LIN {X 0,Y 523.908,Z 265.034,A -85,B 0,C 180,E1 -4736.634,E2 -4736.634} C_VEL
LIN {X 0,Y 523.939,Z 265.035,A -85,B 0,C 180,E1 -4739.356,E2 -4739.356} C_VEL
LIN {X 0,Y 523.937,Z 265.029,A -85,B 0,C 180,E1 -4742.29,E2 -4742.29} C_VEL
LIN {X 0,Y 523.899,Z 265.041,A -85,B 0,C 180,E1 -4745.427,E2 -4745.427} C_VEL
LIN {X 0,Y 523.983,Z 265.186,A -85,B 0,C 180,E1 -4747.547,E2 -4747.547} C_VEL
LIN {X 0,Y 524.776,Z 271.643,A -85,B 0,C 180,E1 -4748.803,E2 -4748.803} C_VEL
LIN {X 0,Y 524.426,Z 286.9,A -85,B 0,C 180,E1 -4751.644,E2 -4751.644} C_VEL
LIN {X 0,Y 524.115,Z 304.678,A -85,B 0,C 180,E1 -4754.898,E2 -4754.898} C_VEL
LIN {X 0,Y 523.825,Z 322.199,A -85,B 0,C 180,E1 -4758.077,E2 -4758.077} C_VEL
LIN {X 0,Y 524.969,Z 332.235,A -85,B 0,C 180,E1 -4758.254,E2 -4758.254} C_VEL
LIN {X 0,Y 524.703,Z 399.496,A -85,B 0,C 180,E1 -4759.192,E2 -4759.192} C_VEL
LIN {X 0,Y 524.561,Z 409.221,A -85,B 0,C 180,E1 -4759.433,E2 -4759.433} C_VEL
LIN {X 0,Y 524.413,Z 420.832,A -85,B 0,C 180,E1 -4759.869,E2 -4759.869} C_VEL
LIN {X 0,Y 524.207,Z 431.496,A -85,B 0,C 180,E1 -4760.45,E2 -4760.45} C_VEL
LIN {X 0,Y 524.097,Z 439.84,A -85,B 0,C 180,E1 -4761.032,E2 -4761.032} C_VEL
LIN {X 0,Y 523.882,Z 447.732,A -85,B 0,C 180,E1 -4761.708,E2 -4761.708} C_VEL
LIN {X 0,Y 523.71,Z 455.111,A -85,B 0,C 180,E1 -4762.482,E2 -4762.482} C_VEL
LIN {X 0,Y 523.63,Z 462.468,A -85,B 0,C 180,E1 -4763.431,E2 -4763.431} C_VEL
LIN {X 0,Y 523.538,Z 468.474,A -85,B 0,C 180,E1 -4764.415,E2 -4764.415} C_VEL
LIN {X 0,Y 523.406,Z 473.097,A -85,B 0,C 180,E1 -4765.379,E2 -4765.379} C_VEL
LIN {X 0,Y 523.454,Z 476.104,A -85,B 0,C 180,E1 -4766.151,E2 -4766.151} C_VEL
LIN {X 0,Y 523.379,Z 478.431,A -85,B 0,C 180,E1 -4766.921,E2 -4766.921} C_VEL
LIN {X 0,Y 523.336,Z 480.183,A -85,B 0,C 180,E1 -4767.691,E2 -4767.691} C_VEL
LIN {X 0,Y 523.273,Z 481.437,A -85,B 0,C 180,E1 -4768.461,E2 -4768.461} C_VEL
LIN {X 0,Y 523.247,Z 482.217,A -85,B 0,C 180,E1 -4769.23,E2 -4769.23} C_VEL
LIN {X 0,Y 523.246,Z 482.512,A -85,B 0,C 180,E1 -4770,E2 -4770} C_VEL
LIN {X 0,Y 523.247,Z 482.215,A -85,B 0,C 180,E1 -4770.77,E2 -4770.77} C_VEL
LIN {X 0,Y 523.273,Z 481.433,A -85,B 0,C 180,E1 -4771.539,E2 -4771.539} C_VEL
LIN {X 0,Y 523.336,Z 480.177,A -85,B 0,C 180,E1 -4772.309,E2 -4772.309} C_VEL
LIN {X 0,Y 523.407,Z 477.267,A -85,B 0,C 180,E1 -4773.464,E2 -4773.464} C_VEL
LIN {X 0,Y 523.454,Z 474.613,A -85,B 0,C 180,E1 -4774.235,E2 -4774.235} C_VEL
LIN {X 0,Y 523.484,Z 469.419,A -85,B 0,C 180,E1 -4775.392,E2 -4775.392} C_VEL
LIN {X 0,Y 523.596,Z 463.434,A -85,B 0,C 180,E1 -4776.422,E2 -4776.422} C_VEL
LIN {X 0,Y 523.698,Z 456.795,A -85,B 0,C 180,E1 -4777.324,E2 -4777.324} C_VEL
LIN {X 0,Y 523.856,Z 448.738,A -85,B 0,C 180,E1 -4778.195,E2 -4778.195} C_VEL
LIN {X 0,Y 524.08,Z 441.048,A -85,B 0,C 180,E1 -4778.871,E2 -4778.871} C_VEL
LIN {X 0,Y 524.198,Z 432.968,A -85,B 0,C 180,E1 -4779.453,E2 -4779.453} C_VEL
LIN {X 0,Y 524.337,Z 424.594,A -85,B 0,C 180,E1 -4779.937,E2 -4779.937} C_VEL
LIN {X 0,Y 524.502,Z 416.045,A -85,B 0,C 180,E1 -4780.324,E2 -4780.324} C_VEL
LIN {X 0,Y 524.571,Z 405.846,A -85,B 0,C 180,E1 -4780.664,E2 -4780.664} C_VEL
LIN {X 0,Y 524.779,Z 393.965,A -85,B 0,C 180,E1 -4780.904,E2 -4780.904} C_VEL
LIN {X 0,Y 524.782,Z 329.722,A -85,B 0,C 180,E1 -4781.784,E2 -4781.784} C_VEL
LIN {X 0,Y 523.821,Z 322.037,A -85,B 0,C 180,E1 -4781.93,E2 -4781.93} C_VEL
LIN {X 0,Y 524.082,Z 303.651,A -85,B 0,C 180,E1 -4785.231,E2 -4785.231} C_VEL
LIN {X 0,Y 524.369,Z 287.56,A -85,B 0,C 180,E1 -4788.156,E2 -4788.156} C_VEL
LIN {X 0,Y 524.64,Z 270.939,A -85,B 0,C 180,E1 -4791.203,E2 -4791.203} C_VEL
LIN {X 0,Y 523.965,Z 265.034,A -85,B 0,C 180,E1 -4792.349,E2 -4792.349} C_VEL
LIN {X 0,Y 523.896,Z 265.035,A -85,B 0,C 180,E1 -4795.421,E2 -4795.421} C_VEL
LIN {X 0,Y 523.906,Z 265.034,A -85,B 0,C 180,E1 -4798.002,E2 -4798.002} C_VEL
LIN {X 0,Y 523.93,Z 265.037,A -85,B 0,C 180,E1 -4800.852,E2 -4800.852} C_VEL
LIN {X 0,Y 523.924,Z 265.03,A -85,B 0,C 180,E1 -4803.729,E2 -4803.729} C_VEL
LIN {X 0,Y 523.897,Z 265.035,A -85,B 0,C 180,E1 -4806.4,E2 -4806.4} C_VEL
LIN {X 0,Y 523.913,Z 265.041,A -85,B 0,C 180,E1 -4809.084,E2 -4809.084} C_VEL
LIN {X 0,Y 523.931,Z 265.029,A -85,B 0,C 180,E1 -4812.119,E2 -4812.119} C_VEL
LIN {X 0,Y 523.941,Z 265.037,A -85,B 0,C 180,E1 -4815.309,E2 -4815.309} C_VEL
LIN {X 0,Y 523.95,Z 265.026,A -85,B 0,C 180,E1 -4818.689,E2 -4818.689} C_VEL
LIN {X 0,Y 523.903,Z 265.035,A -85,B 0,C 180,E1 -4821.08,E2 -4821.08} C_VEL
LIN {X 0,Y 523.913,Z 265.038,A -85,B 0,C 180,E1 -4823.826,E2 -4823.826} C_VEL
LIN {X 0,Y 523.93,Z 265.027,A -85,B 0,C 180,E1 -4826.635,E2 -4826.635} C_VEL
LIN {X 0,Y 523.944,Z 265.029,A -85,B 0,C 180,E1 -4829.355,E2 -4829.355} C_VEL
LIN {X 0,Y 523.963,Z 265.026,A -85,B 0,C 180,E1 -4832.281,E2 -4832.281} C_VEL
LIN {X 0,Y 523.933,Z 265.03,A -85,B 0,C 180,E1 -4834.58,E2 -4834.58} C_VEL
LIN {X 0,Y 523.905,Z 265.034,A -85,B 0,C 180,E1 -4837.756,E2 -4837.756} C_VEL
LIN {X 0,Y 523.959,Z 265.032,A -85,B 0,C 180,E1 -4840.407,E2 -4840.407} C_VEL
LIN {X 0,Y 523.949,Z 265.027,A -85,B 0,C 180,E1 -4842.837,E2 -4842.837} C_VEL
LIN {X 0,Y 523.96,Z 265.023,A -85,B 0,C 180,E1 -4845.235,E2 -4845.235} C_VEL
LIN {X 0,Y 523.998,Z 265.028,A -85,B 0,C 180,E1 -4848.394,E2 -4848.394} C_VEL
LIN {X 0,Y 523.988,Z 265.019,A -85,B 0,C 180,E1 -4851.516,E2 -4851.516} C_VEL
LIN {X 0,Y 524.083,Z 265.017,A -85,B 0,C 180,E1 -4854.614,E2 -4854.614} C_VEL
LIN {X 0,Y 524.094,Z 265.006,A -85,B 0,C 180,E1 -4857.694,E2 -4857.694} C_VEL
LIN {X 0,Y 524.11,Z 265.012,A -85,B 0,C 180,E1 -4860.768,E2 -4860.768} C_VEL
LIN {X 0,Y 524.059,Z 265.019,A -85,B 0,C 180,E1 -4863.075,E2 -4863.075} C_VEL
LIN {X 0,Y 524.017,Z 265.017,A -85,B 0,C 180,E1 -4866.159,E2 -4866.159} C_VEL
LIN {X 0,Y 523.991,Z 265.02,A -85,B 0,C 180,E1 -4868.484,E2 -4868.484} C_VEL
LIN {X 0,Y 523.988,Z 265.023,A -85,B 0,C 180,E1 -4871.74,E2 -4871.74} C_VEL
LIN {X 0,Y 523.979,Z 265.026,A -85,B 0,C 180,E1 -4875.053,E2 -4875.053} C_VEL
LIN {X 0,Y 523.951,Z 265.031,A -85,B 0,C 180,E1 -4877.97,E2 -4877.97} C_VEL
LIN {X 0,Y 523.959,Z 265.025,A -85,B 0,C 180,E1 -4880.411,E2 -4880.411} C_VEL
LIN {X 0,Y 523.904,Z 265.033,A -85,B 0,C 180,E1 -4882.894,E2 -4882.894} C_VEL
LIN {X 0,Y 523.943,Z 265.031,A -85,B 0,C 180,E1 -4885.419,E2 -4885.419} C_VEL
LIN {X 0,Y 523.96,Z 265.034,A -85,B 0,C 180,E1 -4888,E2 -4888} C_VEL
LIN {X 0,Y 523.939,Z 265.028,A -85,B 0,C 180,E1 -4890.857,E2 -4890.857} C_VEL
LIN {X 0,Y 523.952,Z 265.03,A -85,B 0,C 180,E1 -4893.736,E2 -4893.736} C_VEL
LIN {X 0,Y 523.916,Z 265.039,A -85,B 0,C 180,E1 -4896.406,E2 -4896.406} C_VEL
LIN {X 0,Y 523.923,Z 265.032,A -85,B 0,C 180,E1 -4899.085,E2 -4899.085} C_VEL
LIN {X 0,Y 523.961,Z 265.027,A -85,B 0,C 180,E1 -4901.313,E2 -4901.313} C_VEL
LIN {X 0,Y 523.942,Z 265.155,A -85,B 0,C 180,E1 -4904.015,E2 -4904.015} C_VEL
LIN {X 0,Y 523.901,Z 277.544,A -85,B 0,C 180,E1 -4906.558,E2 -4906.558} C_VEL
LIN {X 0,Y 523.203,Z 280.386,A -85,B 0,C 180,E1 -4907.119,E2 -4907.119} C_VEL
LIN {X 0,Y 517.424,Z 289.883,A -85,B 0,C 180,E1 -4908.932,E2 -4908.932} C_VEL
LIN {X 0,Y 516.76,Z 292.676,A -85,B 0,C 180,E1 -4909.507,E2 -4909.507} C_VEL
LIN {X 0,Y 516.771,Z 294.884,A -85,B 0,C 180,E1 -4909.971,E2 -4909.971} C_VEL
LIN {X 0,Y 518.022,Z 305.126,A -85,B 0,C 180,E1 -4910.155,E2 -4910.155} C_VEL
LIN {X 0,Y 517.74,Z 371.268,A -85,B 0,C 180,E1 -4911.094,E2 -4911.094} C_VEL
LIN {X 0,Y 517.645,Z 381.412,A -85,B 0,C 180,E1 -4911.353,E2 -4911.353} C_VEL
LIN {X 0,Y 517.507,Z 392.694,A -85,B 0,C 180,E1 -4911.791,E2 -4911.791} C_VEL
LIN {X 0,Y 517.283,Z 402.236,A -85,B 0,C 180,E1 -4912.312,E2 -4912.312} C_VEL
LIN {X 0,Y 517.132,Z 410.829,A -85,B 0,C 180,E1 -4912.911,E2 -4912.911} C_VEL
LIN {X 0,Y 516.91,Z 418.134,A -85,B 0,C 180,E1 -4913.534,E2 -4913.534} C_VEL
LIN {X 0,Y 516.803,Z 424.755,A -85,B 0,C 180,E1 -4914.216,E2 -4914.216} C_VEL
LIN {X 0,Y 516.67,Z 430.573,A -85,B 0,C 180,E1 -4914.929,E2 -4914.929} C_VEL
LIN {X 0,Y 516.515,Z 436.787,A -85,B 0,C 180,E1 -4915.857,E2 -4915.857} C_VEL
LIN {X 0,Y 516.448,Z 441.827,A -85,B 0,C 180,E1 -4916.792,E2 -4916.792} C_VEL
LIN {X 0,Y 516.359,Z 446.667,A -85,B 0,C 180,E1 -4917.94,E2 -4917.94} C_VEL
LIN {X 0,Y 516.307,Z 450.049,A -85,B 0,C 180,E1 -4919.044,E2 -4919.044} C_VEL
LIN {X 0,Y 516.239,Z 451.555,A -85,B 0,C 180,E1 -4919.755,E2 -4919.755} C_VEL
LIN {X 0,Y 516.219,Z 452.9,A -85,B 0,C 180,E1 -4920.653,E2 -4920.653} C_VEL
LIN {X 0,Y 516.174,Z 453.582,A -85,B 0,C 180,E1 -4921.541,E2 -4921.541} C_VEL
LIN {X 0,Y 516.179,Z 453.632,A -85,B 0,C 180,E1 -4922.425,E2 -4922.425} C_VEL
LIN {X 0,Y 516.182,Z 453.064,A -85,B 0,C 180,E1 -4923.302,E2 -4923.302} C_VEL
LIN {X 0,Y 516.186,Z 451.886,A -85,B 0,C 180,E1 -4924.172,E2 -4924.172} C_VEL
LIN {X 0,Y 516.267,Z 450.057,A -85,B 0,C 180,E1 -4925.04,E2 -4925.04} C_VEL
LIN {X 0,Y 516.336,Z 447.541,A -85,B 0,C 180,E1 -4925.9,E2 -4925.9} C_VEL
LIN {X 0,Y 516.409,Z 442.393,A -85,B 0,C 180,E1 -4927.179,E2 -4927.179} C_VEL
LIN {X 0,Y 516.515,Z 437.678,A -85,B 0,C 180,E1 -4928.08,E2 -4928.08} C_VEL
LIN {X 0,Y 516.606,Z 432.66,A -85,B 0,C 180,E1 -4928.869,E2 -4928.869} C_VEL
LIN {X 0,Y 516.736,Z 427.232,A -85,B 0,C 180,E1 -4929.585,E2 -4929.585} C_VEL
LIN {X 0,Y 516.891,Z 420.375,A -85,B 0,C 180,E1 -4930.336,E2 -4930.336} C_VEL
LIN {X 0,Y 517.035,Z 413.529,A -85,B 0,C 180,E1 -4930.961,E2 -4930.961} C_VEL
LIN {X 0,Y 517.261,Z 405.127,A -85,B 0,C 180,E1 -4931.586,E2 -4931.586} C_VEL
LIN {X 0,Y 517.429,Z 396.432,A -85,B 0,C 180,E1 -4932.102,E2 -4932.102} C_VEL
LIN {X 0,Y 517.564,Z 387.033,A -85,B 0,C 180,E1 -4932.534,E2 -4932.534} C_VEL
LIN {X 0,Y 517.749,Z 376.5,A -85,B 0,C 180,E1 -4932.88,E2 -4932.88} C_VEL
LIN {X 0,Y 517.852,Z 362.604,A -85,B 0,C 180,E1 -4933.137,E2 -4933.137} C_VEL
LIN {X 0,Y 517.873,Z 302.517,A -85,B 0,C 180,E1 -4933.974,E2 -4933.974} C_VEL
LIN {X 0,Y 516.718,Z 295.169,A -85,B 0,C 180,E1 -4934.115,E2 -4934.115} C_VEL
LIN {X 0,Y 516.912,Z 282.012,A -85,B 0,C 180,E1 -4937.037,E2 -4937.037} C_VEL
LIN {X 0,Y 517.088,Z 269.588,A -85,B 0,C 180,E1 -4939.823,E2 -4939.823} C_VEL
LIN {X 0,Y 516.99,Z 265.9,A -85,B 0,C 180,E1 -4940.71,E2 -4940.71} C_VEL
LIN {X 0,Y 517.003,Z 265.901,A -85,B 0,C 180,E1 -4943.757,E2 -4943.757} C_VEL
LIN {X 0,Y 517.013,Z 265.89,A -85,B 0,C 180,E1 -4946.883,E2 -4946.883} C_VEL
LIN {X 0,Y 517.087,Z 265.889,A -85,B 0,C 180,E1 -4950,E2 -4950} C_VEL
LIN {X 0,Y 517.014,Z 265.89,A -85,B 0,C 180,E1 -4953.117,E2 -4953.117} C_VEL
LIN {X 0,Y 516.99,Z 265.901,A -85,B 0,C 180,E1 -4956.243,E2 -4956.243} C_VEL
LIN {X 0,Y 516.967,Z 265.9,A -85,B 0,C 180,E1 -4958.6,E2 -4958.6} C_VEL
LIN {X 0,Y 516.953,Z 265.9,A -85,B 0,C 180,E1 -4961.806,E2 -4961.806} C_VEL
LIN {X 0,Y 516.946,Z 265.899,A -85,B 0,C 180,E1 -4965.146,E2 -4965.146} C_VEL
LIN {X 0,Y 516.917,Z 265.906,A -85,B 0,C 180,E1 -4968.222,E2 -4968.222} C_VEL
LIN {X 0,Y 516.912,Z 265.912,A -85,B 0,C 180,E1 -4970.701,E2 -4970.701} C_VEL
LIN {X 0,Y 516.901,Z 265.905,A -85,B 0,C 180,E1 -4974.072,E2 -4974.072} C_VEL
LIN {X 0,Y 516.922,Z 265.908,A -85,B 0,C 180,E1 -4976.657,E2 -4976.657} C_VEL
LIN {X 0,Y 516.909,Z 265.905,A -85,B 0,C 180,E1 -4979.523,E2 -4979.523} C_VEL
LIN {X 0,Y 516.891,Z 265.907,A -85,B 0,C 180,E1 -4982.542,E2 -4982.542} C_VEL
LIN {X 0,Y 516.861,Z 265.916,A -85,B 0,C 180,E1 -4985.329,E2 -4985.329} C_VEL
LIN {X 0,Y 516.875,Z 265.908,A -85,B 0,C 180,E1 -4987.942,E2 -4987.942} C_VEL
LIN {X 0,Y 516.877,Z 265.908,A -85,B 0,C 180,E1 -4990.741,E2 -4990.741} C_VEL
LIN {X 0,Y 516.877,Z 265.908,A -85,B 0,C 180,E1 -4992.83,E2 -4992.83} C_VEL
LIN {X 0,Y 516.916,Z 265.905,A -85,B 0,C 180,E1 -4995.009,E2 -4995.009} C_VEL
LIN {X 0,Y 516.916,Z 265.903,A -85,B 0,C 180,E1 -4998.397,E2 -4998.397} C_VEL
LIN {X 0,Y 516.879,Z 265.91,A -85,B 0,C 180,E1 -5001.284,E2 -5001.284} C_VEL
LIN {X 0,Y 516.882,Z 265.91,A -85,B 0,C 180,E1 -5004.22,E2 -5004.22} C_VEL
LIN {X 0,Y 516.886,Z 265.906,A -85,B 0,C 180,E1 -5007.052,E2 -5007.052} C_VEL
LIN {X 0,Y 516.891,Z 265.911,A -85,B 0,C 180,E1 -5009.796,E2 -5009.796} C_VEL
LIN {X 0,Y 516.919,Z 265.906,A -85,B 0,C 180,E1 -5012.467,E2 -5012.467} C_VEL
LIN {X 0,Y 516.9,Z 265.904,A -85,B 0,C 180,E1 -5015.071,E2 -5015.071} C_VEL
LIN {X 0,Y 516.874,Z 265.915,A -85,B 0,C 180,E1 -5018.462,E2 -5018.462} C_VEL
LIN {X 0,Y 516.891,Z 265.907,A -85,B 0,C 180,E1 -5020.954,E2 -5020.954} C_VEL
LIN {X 0,Y 516.901,Z 265.904,A -85,B 0,C 180,E1 -5023.41,E2 -5023.41} C_VEL
LIN {X 0,Y 516.882,Z 265.907,A -85,B 0,C 180,E1 -5025.833,E2 -5025.833} C_VEL
LIN {X 0,Y 516.952,Z 265.901,A -85,B 0,C 180,E1 -5028.233,E2 -5028.233} C_VEL
LIN {X 0,Y 516.956,Z 265.899,A -85,B 0,C 180,E1 -5031.399,E2 -5031.399} C_VEL
LIN {X 0,Y 516.989,Z 265.893,A -85,B 0,C 180,E1 -5033.756,E2 -5033.756} C_VEL
LIN {X 0,Y 517.001,Z 265.9,A -85,B 0,C 180,E1 -5036.883,E2 -5036.883} C_VEL
LIN {X 0,Y 517.066,Z 265.883,A -85,B 0,C 180,E1 -5040,E2 -5040} C_VEL
LIN {X 0,Y 517.003,Z 265.9,A -85,B 0,C 180,E1 -5043.117,E2 -5043.117} C_VEL
LIN {X 0,Y 516.988,Z 265.893,A -85,B 0,C 180,E1 -5046.243,E2 -5046.243} C_VEL
LIN {X 0,Y 516.942,Z 265.908,A -85,B 0,C 180,E1 -5049.389,E2 -5049.389} C_VEL
LIN {X 0,Y 516.97,Z 265.9,A -85,B 0,C 180,E1 -5051.824,E2 -5051.824} C_VEL
LIN {X 0,Y 516.93,Z 265.903,A -85,B 0,C 180,E1 -5055.147,E2 -5055.147} C_VEL
LIN {X 0,Y 516.911,Z 265.905,A -85,B 0,C 180,E1 -5058.223,E2 -5058.223} C_VEL
LIN {X 0,Y 516.899,Z 265.904,A -85,B 0,C 180,E1 -5060.702,E2 -5060.702} C_VEL
LIN {X 0,Y 516.899,Z 265.912,A -85,B 0,C 180,E1 -5064.073,E2 -5064.073} C_VEL
LIN {X 0,Y 516.91,Z 265.904,A -85,B 0,C 180,E1 -5066.659,E2 -5066.659} C_VEL
LIN {X 0,Y 516.899,Z 265.905,A -85,B 0,C 180,E1 -5069.524,E2 -5069.524} C_VEL
LIN {X 0,Y 516.884,Z 265.911,A -85,B 0,C 180,E1 -5072.544,E2 -5072.544} C_VEL
LIN {X 0,Y 516.868,Z 265.908,A -85,B 0,C 180,E1 -5075.332,E2 -5075.332} C_VEL
LIN {X 0,Y 516.87,Z 265.91,A -85,B 0,C 180,E1 -5077.944,E2 -5077.944} C_VEL
LIN {X 0,Y 516.875,Z 265.914,A -85,B 0,C 180,E1 -5080.742,E2 -5080.742} C_VEL
LIN {X 0,Y 516.874,Z 265.914,A -85,B 0,C 180,E1 -5082.832,E2 -5082.832} C_VEL
LIN {X 0,Y 516.887,Z 265.911,A -85,B 0,C 180,E1 -5085.008,E2 -5085.008} C_VEL
LIN {X 0,Y 516.895,Z 265.908,A -85,B 0,C 180,E1 -5088.401,E2 -5088.401} C_VEL
LIN {X 0,Y 516.873,Z 265.912,A -85,B 0,C 180,E1 -5091.285,E2 -5091.285} C_VEL
LIN {X 0,Y 516.864,Z 265.909,A -85,B 0,C 180,E1 -5094.22,E2 -5094.22} C_VEL
LIN {X 0,Y 516.876,Z 265.916,A -85,B 0,C 180,E1 -5097.053,E2 -5097.053} C_VEL
LIN {X 0,Y 516.878,Z 265.909,A -85,B 0,C 180,E1 -5099.796,E2 -5099.796} C_VEL
LIN {X 0,Y 516.888,Z 265.907,A -85,B 0,C 180,E1 -5102.466,E2 -5102.466} C_VEL
LIN {X 0,Y 516.869,Z 265.916,A -85,B 0,C 180,E1 -5105.646,E2 -5105.646} C_VEL
LIN {X 0,Y 516.937,Z 265.971,A -85,B 0,C 180,E1 -5107.407,E2 -5107.407} C_VEL
LIN {X 0,Y 517.804,Z 272.574,A -85,B 0,C 180,E1 -5108.712,E2 -5108.712} C_VEL
LIN {X 0,Y 517.383,Z 288.908,A -85,B 0,C 180,E1 -5111.795,E2 -5111.795} C_VEL
LIN {X 0,Y 517.08,Z 305.082,A -85,B 0,C 180,E1 -5114.799,E2 -5114.799} C_VEL
LIN {X 0,Y 516.781,Z 322.075,A -85,B 0,C 180,E1 -5117.924,E2 -5117.924} C_VEL
LIN {X 0,Y 518.034,Z 332.048,A -85,B 0,C 180,E1 -5118.095,E2 -5118.095} C_VEL
LIN {X 0,Y 517.738,Z 399.23,A -85,B 0,C 180,E1 -5119.045,E2 -5119.045} C_VEL
LIN {X 0,Y 517.559,Z 408.98,A -85,B 0,C 180,E1 -5119.289,E2 -5119.289} C_VEL
LIN {X 0,Y 517.455,Z 419.489,A -85,B 0,C 180,E1 -5119.682,E2 -5119.682} C_VEL
LIN {X 0,Y 517.235,Z 429.777,A -85,B 0,C 180,E1 -5120.221,E2 -5120.221} C_VEL
LIN {X 0,Y 517.074,Z 438.396,A -85,B 0,C 180,E1 -5120.811,E2 -5120.811} C_VEL
LIN {X 0,Y 516.878,Z 446.501,A -85,B 0,C 180,E1 -5121.497,E2 -5121.497} C_VEL
LIN {X 0,Y 516.697,Z 453.196,A -85,B 0,C 180,E1 -5122.183,E2 -5122.183} C_VEL
LIN {X 0,Y 516.6,Z 459.552,A -85,B 0,C 180,E1 -5122.967,E2 -5122.967} C_VEL
LIN {X 0,Y 516.522,Z 466.011,A -85,B 0,C 180,E1 -5123.947,E2 -5123.947} C_VEL
LIN {X 0,Y 516.348,Z 471.154,A -85,B 0,C 180,E1 -5124.924,E2 -5124.924} C_VEL
LIN {X 0,Y 516.365,Z 475.906,A -85,B 0,C 180,E1 -5126.098,E2 -5126.098} C_VEL
LIN {X 0,Y 516.294,Z 478.234,A -85,B 0,C 180,E1 -5126.879,E2 -5126.879} C_VEL
LIN {X 0,Y 516.262,Z 479.987,A -85,B 0,C 180,E1 -5127.659,E2 -5127.659} C_VEL
LIN {X 0,Y 516.19,Z 481.241,A -85,B 0,C 180,E1 -5128.44,E2 -5128.44} C_VEL
LIN {X 0,Y 516.157,Z 482.022,A -85,B 0,C 180,E1 -5129.22,E2 -5129.22} C_VEL
LIN {X 0,Y 516.154,Z 482.316,A -85,B 0,C 180,E1 -5130,E2 -5130} C_VEL
LIN {X 0,Y 516.157,Z 482.018,A -85,B 0,C 180,E1 -5130.78,E2 -5130.78} C_VEL
LIN {X 0,Y 516.19,Z 481.236,A -85,B 0,C 180,E1 -5131.56,E2 -5131.56} C_VEL
LIN {X 0,Y 516.262,Z 479.979,A -85,B 0,C 180,E1 -5132.341,E2 -5132.341} C_VEL
LIN {X 0,Y 516.325,Z 477.067,A -85,B 0,C 180,E1 -5133.512,E2 -5133.512} C_VEL
LIN {X 0,Y 516.345,Z 474.411,A -85,B 0,C 180,E1 -5134.293,E2 -5134.293} C_VEL
LIN {X 0,Y 516.429,Z 469.214,A -85,B 0,C 180,E1 -5135.466,E2 -5135.466} C_VEL
LIN {X 0,Y 516.503,Z 463.851,A -85,B 0,C 180,E1 -5136.408,E2 -5136.408} C_VEL
LIN {X 0,Y 516.625,Z 456.582,A -85,B 0,C 180,E1 -5137.425,E2 -5137.425} C_VEL
LIN {X 0,Y 516.821,Z 448.522,A -85,B 0,C 180,E1 -5138.307,E2 -5138.307} C_VEL
LIN {X 0,Y 517.058,Z 440.828,A -85,B 0,C 180,E1 -5138.993,E2 -5138.993} C_VEL
LIN {X 0,Y 517.164,Z 432.742,A -85,B 0,C 180,E1 -5139.582,E2 -5139.582} C_VEL
LIN {X 0,Y 517.331,Z 424.362,A -85,B 0,C 180,E1 -5140.073,E2 -5140.073} C_VEL
LIN {X 0,Y 517.514,Z 415.805,A -85,B 0,C 180,E1 -5140.465,E2 -5140.465} C_VEL
LIN {X 0,Y 517.611,Z 405.593,A -85,B 0,C 180,E1 -5140.809,E2 -5140.809} C_VEL
LIN {X 0,Y 517.825,Z 392.225,A -85,B 0,C 180,E1 -5141.072,E2 -5141.072} C_VEL
LIN {X 0,Y 517.874,Z 330.713,A -85,B 0,C 180,E1 -5141.927,E2 -5141.927} C_VEL
LIN {X 0,Y 516.771,Z 321.808,A -85,B 0,C 180,E1 -5142.099,E2 -5142.099} C_VEL
LIN {X 0,Y 517.034,Z 304.866,A -85,B 0,C 180,E1 -5145.183,E2 -5145.183} C_VEL
LIN {X 0,Y 517.338,Z 288.416,A -85,B 0,C 180,E1 -5148.207,E2 -5148.207} C_VEL
LIN {X 0,Y 517.634,Z 272.903,A -85,B 0,C 180,E1 -5151.087,E2 -5151.087} C_VEL
LIN {X 0,Y 517.327,Z 268.449,A -85,B 0,C 180,E1 -5151.937,E2 -5151.937} C_VEL
LIN {X 0,Y 516.927,Z 265.911,A -85,B 0,C 180,E1 -5152.47,E2 -5152.47} C_VEL
LIN {X 0,Y 516.869,Z 265.911,A -85,B 0,C 180,E1 -5155.792,E2 -5155.792} C_VEL
LIN {X 0,Y 516.847,Z 265.918,A -85,B 0,C 180,E1 -5158.419,E2 -5158.419} C_VEL
LIN {X 0,Y 516.882,Z 265.912,A -85,B 0,C 180,E1 -5161.109,E2 -5161.109} C_VEL
LIN {X 0,Y 516.88,Z 265.908,A -85,B 0,C 180,E1 -5163.961,E2 -5163.961} C_VEL
LIN {X 0,Y 516.87,Z 265.915,A -85,B 0,C 180,E1 -5166.745,E2 -5166.745} C_VEL
LIN {X 0,Y 516.875,Z 265.911,A -85,B 0,C 180,E1 -5169.721,E2 -5169.721} C_VEL
LIN {X 0,Y 516.894,Z 265.908,A -85,B 0,C 180,E1 -5171.775,E2 -5171.775} C_VEL
LIN {X 0,Y 516.887,Z 265.913,A -85,B 0,C 180,E1 -5175.006,E2 -5175.006} C_VEL
LIN {X 0,Y 516.906,Z 265.903,A -85,B 0,C 180,E1 -5178.398,E2 -5178.398} C_VEL
LIN {X 0,Y 516.868,Z 265.914,A -85,B 0,C 180,E1 -5181.283,E2 -5181.283} C_VEL
LIN {X 0,Y 516.876,Z 265.909,A -85,B 0,C 180,E1 -5184.22,E2 -5184.22} C_VEL
LIN {X 0,Y 516.883,Z 265.906,A -85,B 0,C 180,E1 -5187.052,E2 -5187.052} C_VEL
LIN {X 0,Y 516.88,Z 265.915,A -85,B 0,C 180,E1 -5189.796,E2 -5189.796} C_VEL
LIN {X 0,Y 516.912,Z 265.902,A -85,B 0,C 180,E1 -5192.467,E2 -5192.467} C_VEL
LIN {X 0,Y 516.862,Z 265.909,A -85,B 0,C 180,E1 -5195.069,E2 -5195.069} C_VEL
LIN {X 0,Y 516.855,Z 265.911,A -85,B 0,C 180,E1 -5197.621,E2 -5197.621} C_VEL
LIN {X 0,Y 516.917,Z 265.909,A -85,B 0,C 180,E1 -5200.129,E2 -5200.129} C_VEL
LIN {X 0,Y 516.905,Z 265.907,A -85,B 0,C 180,E1 -5202.595,E2 -5202.595} C_VEL
LIN {X 0,Y 516.926,Z 265.9,A -85,B 0,C 180,E1 -5205.03,E2 -5205.03} C_VEL
LIN {X 0,Y 516.951,Z 265.903,A -85,B 0,C 180,E1 -5208.233,E2 -5208.233} C_VEL
LIN {X 0,Y 516.954,Z 265.895,A -85,B 0,C 180,E1 -5211.4,E2 -5211.4} C_VEL
LIN {X 0,Y 516.987,Z 265.893,A -85,B 0,C 180,E1 -5213.757,E2 -5213.757} C_VEL
LIN {X 0,Y 517.002,Z 265.897,A -85,B 0,C 180,E1 -5216.883,E2 -5216.883} C_VEL
LIN {X 0,Y 517.066,Z 265.883,A -85,B 0,C 180,E1 -5220,E2 -5220} C_VEL
LIN {X 0,Y 517.001,Z 265.898,A -85,B 0,C 180,E1 -5223.117,E2 -5223.117} C_VEL
LIN {X 0,Y 516.979,Z 265.894,A -85,B 0,C 180,E1 -5226.244,E2 -5226.244} C_VEL
LIN {X 0,Y 516.955,Z 265.897,A -85,B 0,C 180,E1 -5228.601,E2 -5228.601} C_VEL
LIN {X 0,Y 516.938,Z 265.9,A -85,B 0,C 180,E1 -5231.807,E2 -5231.807} C_VEL
LIN {X 0,Y 516.931,Z 265.906,A -85,B 0,C 180,E1 -5235.147,E2 -5235.147} C_VEL
LIN {X 0,Y 516.912,Z 265.906,A -85,B 0,C 180,E1 -5238.223,E2 -5238.223} C_VEL
LIN {X 0,Y 516.899,Z 265.904,A -85,B 0,C 180,E1 -5240.702,E2 -5240.702} C_VEL
LIN {X 0,Y 516.899,Z 265.911,A -85,B 0,C 180,E1 -5244.073,E2 -5244.073} C_VEL
LIN {X 0,Y 516.918,Z 265.903,A -85,B 0,C 180,E1 -5246.658,E2 -5246.658} C_VEL
LIN {X 0,Y 516.909,Z 265.906,A -85,B 0,C 180,E1 -5249.526,E2 -5249.526} C_VEL
LIN {X 0,Y 516.887,Z 265.91,A -85,B 0,C 180,E1 -5252.545,E2 -5252.545} C_VEL
LIN {X 0,Y 516.874,Z 265.907,A -85,B 0,C 180,E1 -5255.333,E2 -5255.333} C_VEL
LIN {X 0,Y 516.874,Z 265.913,A -85,B 0,C 180,E1 -5257.944,E2 -5257.944} C_VEL
LIN {X 0,Y 516.895,Z 265.912,A -85,B 0,C 180,E1 -5260.741,E2 -5260.741} C_VEL
LIN {X 0,Y 516.911,Z 265.908,A -85,B 0,C 180,E1 -5263.945,E2 -5263.945} C_VEL
LIN {X 0,Y 516.851,Z 278.942,A -85,B 0,C 180,E1 -5266.638,E2 -5266.638} C_VEL
LIN {X 0,Y 516.76,Z 292.676,A -85,B 0,C 180,E1 -5269.507,E2 -5269.507} C_VEL
LIN {X 0,Y 516.381,Z 294.396,A -85,B 0,C 180,E1 -5269.73,E2 -5269.73} C_VEL
LIN {X 0,Y 515.17,Z 297.475,A -85,B 0,C 180,E1 -5269.907,E2 -5269.907} C_VEL
LIN {X 0,Y 513.228,Z 301.968,A -85,B 0,C 180,E1 -5269.994,E2 -5269.994} C_VEL
LIN {X 0,Y 511.484,Z 307.907,A -85,B 0,C 180,E1 -5270.035,E2 -5270.035} C_VEL
LIN {X 0,Y 510.915,Z 314.38,A -85,B 0,C 180,E1 -5270.112,E2 -5270.112} C_VEL
LIN {X 0,Y 510.998,Z 323.083,A -85,B 0,C 180,E1 -5270.24,E2 -5270.24} C_VEL
LIN {X 0,Y 510.783,Z 371.331,A -85,B 0,C 180,E1 -5270.942,E2 -5270.942} C_VEL
LIN {X 0,Y 510.688,Z 381.454,A -85,B 0,C 180,E1 -5271.203,E2 -5271.203} C_VEL
LIN {X 0,Y 510.552,Z 392.084,A -85,B 0,C 180,E1 -5271.613,E2 -5271.613} C_VEL
LIN {X 0,Y 510.292,Z 402.813,A -85,B 0,C 180,E1 -5272.204,E2 -5272.204} C_VEL
LIN {X 0,Y 510.115,Z 411.178,A -85,B 0,C 180,E1 -5272.798,E2 -5272.798} C_VEL
LIN {X 0,Y 509.885,Z 418.58,A -85,B 0,C 180,E1 -5273.442,E2 -5273.442} C_VEL
LIN {X 0,Y 509.763,Z 424.69,A -85,B 0,C 180,E1 -5274.077,E2 -5274.077} C_VEL
LIN {X 0,Y 509.623,Z 430.895,A -85,B 0,C 180,E1 -5274.849,E2 -5274.849} C_VEL
LIN {X 0,Y 509.46,Z 435.723,A -85,B 0,C 180,E1 -5275.558,E2 -5275.558} C_VEL
LIN {X 0,Y 509.394,Z 440.997,A -85,B 0,C 180,E1 -5276.506,E2 -5276.506} C_VEL
LIN {X 0,Y 509.277,Z 445.174,A -85,B 0,C 180,E1 -5277.44,E2 -5277.44} C_VEL
LIN {X 0,Y 509.259,Z 448.438,A -85,B 0,C 180,E1 -5278.372,E2 -5278.372} C_VEL
LIN {X 0,Y 509.204,Z 450.874,A -85,B 0,C 180,E1 -5279.292,E2 -5279.292} C_VEL
LIN {X 0,Y 509.121,Z 452.839,A -85,B 0,C 180,E1 -5280.42,E2 -5280.42} C_VEL
LIN {X 0,Y 509.09,Z 453.604,A -85,B 0,C 180,E1 -5281.108,E2 -5281.108} C_VEL
LIN {X 0,Y 509.082,Z 453.957,A -85,B 0,C 180,E1 -5282.072,E2 -5282.072} C_VEL
LIN {X 0,Y 509.073,Z 453.637,A -85,B 0,C 180,E1 -5282.899,E2 -5282.899} C_VEL
LIN {X 0,Y 509.083,Z 452.663,A -85,B 0,C 180,E1 -5283.811,E2 -5283.811} C_VEL
LIN {X 0,Y 509.201,Z 450.187,A -85,B 0,C 180,E1 -5285.106,E2 -5285.106} C_VEL
LIN {X 0,Y 509.273,Z 447.532,A -85,B 0,C 180,E1 -5286.017,E2 -5286.017} C_VEL
LIN {X 0,Y 509.333,Z 442.475,A -85,B 0,C 180,E1 -5287.273,E2 -5287.273} C_VEL
LIN {X 0,Y 509.439,Z 438.055,A -85,B 0,C 180,E1 -5288.132,E2 -5288.132} C_VEL
LIN {X 0,Y 509.562,Z 432.683,A -85,B 0,C 180,E1 -5288.987,E2 -5288.987} C_VEL
LIN {X 0,Y 509.691,Z 426.167,A -85,B 0,C 180,E1 -5289.836,E2 -5289.836} C_VEL
LIN {X 0,Y 509.909,Z 419.232,A -85,B 0,C 180,E1 -5290.579,E2 -5290.579} C_VEL
LIN {X 0,Y 510.077,Z 412.114,A -85,B 0,C 180,E1 -5291.213,E2 -5291.213} C_VEL
LIN {X 0,Y 510.281,Z 404.912,A -85,B 0,C 180,E1 -5291.743,E2 -5291.743} C_VEL
LIN {X 0,Y 510.444,Z 396.787,A -85,B 0,C 180,E1 -5292.231,E2 -5292.231} C_VEL
LIN {X 0,Y 510.588,Z 388.311,A -85,B 0,C 180,E1 -5292.632,E2 -5292.632} C_VEL
LIN {X 0,Y 510.739,Z 378.549,A -85,B 0,C 180,E1 -5292.973,E2 -5292.973} C_VEL
LIN {X 0,Y 510.855,Z 368.109,A -85,B 0,C 180,E1 -5293.208,E2 -5293.208} C_VEL
LIN {X 0,Y 511.058,Z 304.087,A -85,B 0,C 180,E1 -5294.116,E2 -5294.116} C_VEL
LIN {X 0,Y 509.709,Z 295.317,A -85,B 0,C 180,E1 -5294.285,E2 -5294.285} C_VEL
LIN {X 0,Y 509.882,Z 282.067,A -85,B 0,C 180,E1 -5297.26,E2 -5297.26} C_VEL
LIN {X 0,Y 510.084,Z 269.621,A -85,B 0,C 180,E1 -5300.083,E2 -5300.083} C_VEL
LIN {X 0,Y 509.941,Z 266.778,A -85,B 0,C 180,E1 -5300.781,E2 -5300.781} C_VEL
LIN {X 0,Y 509.955,Z 266.779,A -85,B 0,C 180,E1 -5303.67,E2 -5303.67} C_VEL
LIN {X 0,Y 510.055,Z 266.763,A -85,B 0,C 180,E1 -5307.631,E2 -5307.631} C_VEL
LIN {X 0,Y 510.065,Z 266.756,A -85,B 0,C 180,E1 -5310.789,E2 -5310.789} C_VEL
LIN {X 0,Y 509.956,Z 266.769,A -85,B 0,C 180,E1 -5313.16,E2 -5313.16} C_VEL
LIN {X 0,Y 509.938,Z 266.778,A -85,B 0,C 180,E1 -5316.33,E2 -5316.33} C_VEL
LIN {X 0,Y 509.913,Z 266.777,A -85,B 0,C 180,E1 -5318.72,E2 -5318.72} C_VEL
LIN {X 0,Y 509.906,Z 266.779,A -85,B 0,C 180,E1 -5321.931,E2 -5321.931} C_VEL
LIN {X 0,Y 509.895,Z 266.777,A -85,B 0,C 180,E1 -5325.241,E2 -5325.241} C_VEL
LIN {X 0,Y 509.868,Z 266.782,A -85,B 0,C 180,E1 -5327.993,E2 -5327.993} C_VEL
LIN {X 0,Y 509.886,Z 266.784,A -85,B 0,C 180,E1 -5330.401,E2 -5330.401} C_VEL
LIN {X 0,Y 509.829,Z 266.785,A -85,B 0,C 180,E1 -5333.563,E2 -5333.563} C_VEL
LIN {X 0,Y 509.909,Z 266.778,A -85,B 0,C 180,E1 -5336.377,E2 -5336.377} C_VEL
LIN {X 0,Y 509.875,Z 266.788,A -85,B 0,C 180,E1 -5338.843,E2 -5338.843} C_VEL
LIN {X 0,Y 509.817,Z 266.788,A -85,B 0,C 180,E1 -5341.589,E2 -5341.589} C_VEL
LIN {X 0,Y 509.834,Z 266.785,A -85,B 0,C 180,E1 -5344.414,E2 -5344.414} C_VEL
LIN {X 0,Y 509.812,Z 266.795,A -85,B 0,C 180,E1 -5347.34,E2 -5347.34} C_VEL
LIN {X 0,Y 509.832,Z 266.784,A -85,B 0,C 180,E1 -5350.381,E2 -5350.381} C_VEL
LIN {X 0,Y 509.817,Z 266.79,A -85,B 0,C 180,E1 -5353.061,E2 -5353.061} C_VEL
LIN {X 0,Y 509.825,Z 266.791,A -85,B 0,C 180,E1 -5355.791,E2 -5355.791} C_VEL
LIN {X 0,Y 509.858,Z 266.781,A -85,B 0,C 180,E1 -5358.575,E2 -5358.575} C_VEL
LIN {X 0,Y 509.844,Z 266.793,A -85,B 0,C 180,E1 -5361.785,E2 -5361.785} C_VEL
LIN {X 0,Y 509.837,Z 266.784,A -85,B 0,C 180,E1 -5364.622,E2 -5364.622} C_VEL
LIN {X 0,Y 509.853,Z 266.785,A -85,B 0,C 180,E1 -5367.48,E2 -5367.48} C_VEL
LIN {X 0,Y 509.872,Z 266.786,A -85,B 0,C 180,E1 -5370.268,E2 -5370.268} C_VEL
LIN {X 0,Y 509.877,Z 266.779,A -85,B 0,C 180,E1 -5372.944,E2 -5372.944} C_VEL
LIN {X 0,Y 509.859,Z 266.782,A -85,B 0,C 180,E1 -5375.573,E2 -5375.573} C_VEL
LIN {X 0,Y 509.838,Z 266.785,A -85,B 0,C 180,E1 -5378.998,E2 -5378.998} C_VEL
LIN {X 0,Y 509.876,Z 266.782,A -85,B 0,C 180,E1 -5381.999,E2 -5381.999} C_VEL
LIN {X 0,Y 509.897,Z 266.782,A -85,B 0,C 180,E1 -5384.818,E2 -5384.818} C_VEL
LIN {X 0,Y 509.887,Z 266.78,A -85,B 0,C 180,E1 -5388.124,E2 -5388.124} C_VEL
LIN {X 0,Y 509.903,Z 266.778,A -85,B 0,C 180,E1 -5391.279,E2 -5391.279} C_VEL
LIN {X 0,Y 509.94,Z 266.771,A -85,B 0,C 180,E1 -5393.67,E2 -5393.67} C_VEL
LIN {X 0,Y 509.944,Z 266.778,A -85,B 0,C 180,E1 -5396.84,E2 -5396.84} C_VEL
LIN {X 0,Y 510.051,Z 266.765,A -85,B 0,C 180,E1 -5399.21,E2 -5399.21} C_VEL
LIN {X 0,Y 509.918,Z 266.777,A -85,B 0,C 180,E1 -5401.579,E2 -5401.579} C_VEL
LIN {X 0,Y 509.945,Z 266.78,A -85,B 0,C 180,E1 -5403.16,E2 -5403.16} C_VEL
LIN {X 0,Y 509.94,Z 266.771,A -85,B 0,C 180,E1 -5406.33,E2 -5406.33} C_VEL
LIN {X 0,Y 509.901,Z 266.777,A -85,B 0,C 180,E1 -5408.72,E2 -5408.72} C_VEL
LIN {X 0,Y 509.938,Z 266.775,A -85,B 0,C 180,E1 -5411.931,E2 -5411.931} C_VEL
LIN {X 0,Y 509.88,Z 266.782,A -85,B 0,C 180,E1 -5415.242,E2 -5415.242} C_VEL
LIN {X 0,Y 509.875,Z 266.785,A -85,B 0,C 180,E1 -5418.001,E2 -5418.001} C_VEL
LIN {X 0,Y 509.837,Z 266.784,A -85,B 0,C 180,E1 -5421.002,E2 -5421.002} C_VEL
LIN {X 0,Y 509.857,Z 266.784,A -85,B 0,C 180,E1 -5424.427,E2 -5424.427} C_VEL
LIN {X 0,Y 509.87,Z 266.78,A -85,B 0,C 180,E1 -5427.056,E2 -5427.056} C_VEL
LIN {X 0,Y 509.846,Z 266.786,A -85,B 0,C 180,E1 -5429.752,E2 -5429.752} C_VEL
LIN {X 0,Y 509.862,Z 266.783,A -85,B 0,C 180,E1 -5432.775,E2 -5432.775} C_VEL
LIN {X 0,Y 509.828,Z 266.785,A -85,B 0,C 180,E1 -5435.581,E2 -5435.581} C_VEL
LIN {X 0,Y 509.839,Z 266.792,A -85,B 0,C 180,E1 -5438.339,E2 -5438.339} C_VEL
LIN {X 0,Y 509.848,Z 266.783,A -85,B 0,C 180,E1 -5441.426,E2 -5441.426} C_VEL
LIN {X 0,Y 509.831,Z 266.795,A -85,B 0,C 180,E1 -5444.671,E2 -5444.671} C_VEL
LIN {X 0,Y 509.838,Z 266.785,A -85,B 0,C 180,E1 -5448.106,E2 -5448.106} C_VEL
LIN {X 0,Y 509.839,Z 266.789,A -85,B 0,C 180,E1 -5450.648,E2 -5450.648} C_VEL
LIN {X 0,Y 509.818,Z 266.787,A -85,B 0,C 180,E1 -5453.648,E2 -5453.648} C_VEL
LIN {X 0,Y 509.836,Z 266.786,A -85,B 0,C 180,E1 -5456.539,E2 -5456.539} C_VEL
LIN {X 0,Y 509.836,Z 266.792,A -85,B 0,C 180,E1 -5459.335,E2 -5459.335} C_VEL
LIN {X 0,Y 509.842,Z 266.785,A -85,B 0,C 180,E1 -5462.052,E2 -5462.052} C_VEL
LIN {X 0,Y 509.799,Z 266.791,A -85,B 0,C 180,E1 -5464.701,E2 -5464.701} C_VEL
LIN {X 0,Y 509.923,Z 266.938,A -85,B 0,C 180,E1 -5467.301,E2 -5467.301} C_VEL
LIN {X 0,Y 510.818,Z 273.499,A -85,B 0,C 180,E1 -5468.618,E2 -5468.618} C_VEL
LIN {X 0,Y 510.415,Z 288.748,A -85,B 0,C 180,E1 -5471.538,E2 -5471.538} C_VEL
LIN {X 0,Y 510.031,Z 305.518,A -85,B 0,C 180,E1 -5474.702,E2 -5474.702} C_VEL
LIN {X 0,Y 509.743,Z 322.03,A -85,B 0,C 180,E1 -5477.759,E2 -5477.759} C_VEL
LIN {X 0,Y 511.073,Z 333.809,A -85,B 0,C 180,E1 -5477.958,E2 -5477.958} C_VEL
LIN {X 0,Y 510.777,Z 398.964,A -85,B 0,C 180,E1 -5478.894,E2 -5478.894} C_VEL
LIN {X 0,Y 510.567,Z 408.738,A -85,B 0,C 180,E1 -5479.14,E2 -5479.14} C_VEL
LIN {X 0,Y 510.449,Z 420.386,A -85,B 0,C 180,E1 -5479.589,E2 -5479.589} C_VEL
LIN {X 0,Y 510.188,Z 431.066,A -85,B 0,C 180,E1 -5480.185,E2 -5480.185} C_VEL
LIN {X 0,Y 510.009,Z 439.417,A -85,B 0,C 180,E1 -5480.782,E2 -5480.782} C_VEL
LIN {X 0,Y 509.813,Z 447.317,A -85,B 0,C 180,E1 -5481.478,E2 -5481.478} C_VEL
LIN {X 0,Y 509.593,Z 454.701,A -85,B 0,C 180,E1 -5482.272,E2 -5482.272} C_VEL
LIN {X 0,Y 509.471,Z 462.572,A -85,B 0,C 180,E1 -5483.323,E2 -5483.323} C_VEL
LIN {X 0,Y 509.348,Z 469.037,A -85,B 0,C 180,E1 -5484.458,E2 -5484.458} C_VEL
LIN {X 0,Y 509.239,Z 474.226,A -85,B 0,C 180,E1 -5485.647,E2 -5485.647} C_VEL
LIN {X 0,Y 509.245,Z 476.881,A -85,B 0,C 180,E1 -5486.44,E2 -5486.44} C_VEL
LIN {X 0,Y 509.191,Z 479.791,A -85,B 0,C 180,E1 -5487.627,E2 -5487.627} C_VEL
LIN {X 0,Y 509.111,Z 481.046,A -85,B 0,C 180,E1 -5488.418,E2 -5488.418} C_VEL
LIN {X 0,Y 509.071,Z 481.826,A -85,B 0,C 180,E1 -5489.209,E2 -5489.209} C_VEL
LIN {X 0,Y 509.065,Z 482.12,A -85,B 0,C 180,E1 -5490,E2 -5490} C_VEL
LIN {X 0,Y 509.071,Z 481.822,A -85,B 0,C 180,E1 -5490.791,E2 -5490.791} C_VEL
LIN {X 0,Y 509.111,Z 481.038,A -85,B 0,C 180,E1 -5491.582,E2 -5491.582} C_VEL
LIN {X 0,Y 509.191,Z 479.781,A -85,B 0,C 180,E1 -5492.373,E2 -5492.373} C_VEL
LIN {X 0,Y 509.245,Z 476.866,A -85,B 0,C 180,E1 -5493.56,E2 -5493.56} C_VEL
LIN {X 0,Y 509.239,Z 474.208,A -85,B 0,C 180,E1 -5494.353,E2 -5494.353} C_VEL
LIN {X 0,Y 509.348,Z 469.009,A -85,B 0,C 180,E1 -5495.542,E2 -5495.542} C_VEL
LIN {X 0,Y 509.468,Z 462.554,A -85,B 0,C 180,E1 -5496.674,E2 -5496.674} C_VEL
LIN {X 0,Y 509.592,Z 454.666,A -85,B 0,C 180,E1 -5497.728,E2 -5497.728} C_VEL
LIN {X 0,Y 509.813,Z 447.281,A -85,B 0,C 180,E1 -5498.522,E2 -5498.522} C_VEL
LIN {X 0,Y 510.009,Z 439.371,A -85,B 0,C 180,E1 -5499.218,E2 -5499.218} C_VEL
LIN {X 0,Y 510.19,Z 431.011,A -85,B 0,C 180,E1 -5499.815,E2 -5499.815} C_VEL
LIN {X 0,Y 510.41,Z 420.325,A -85,B 0,C 180,E1 -5500.411,E2 -5500.411} C_VEL
LIN {X 0,Y 510.579,Z 408.666,A -85,B 0,C 180,E1 -5500.859,E2 -5500.859} C_VEL
LIN {X 0,Y 510.788,Z 398.875,A -85,B 0,C 180,E1 -5501.106,E2 -5501.106} C_VEL
LIN {X 0,Y 510.988,Z 331.768,A -85,B 0,C 180,E1 -5502.072,E2 -5502.072} C_VEL
LIN {X 0,Y 509.691,Z 321.6,A -85,B 0,C 180,E1 -5502.27,E2 -5502.27} C_VEL
LIN {X 0,Y 509.982,Z 305.303,A -85,B 0,C 180,E1 -5505.278,E2 -5505.278} C_VEL
LIN {X 0,Y 510.288,Z 289.933,A -85,B 0,C 180,E1 -5508.138,E2 -5508.138} C_VEL
LIN {X 0,Y 510.636,Z 274.886,A -85,B 0,C 180,E1 -5510.967,E2 -5510.967} C_VEL
LIN {X 0,Y 510.477,Z 270.431,A -85,B 0,C 180,E1 -5511.821,E2 -5511.821} C_VEL
LIN {X 0,Y 509.886,Z 266.788,A -85,B 0,C 180,E1 -5512.558,E2 -5512.558} C_VEL
LIN {X 0,Y 509.799,Z 266.793,A -85,B 0,C 180,E1 -5515.299,E2 -5515.299} C_VEL
LIN {X 0,Y 509.817,Z 266.79,A -85,B 0,C 180,E1 -5518.084,E2 -5518.084} C_VEL
LIN {X 0,Y 509.829,Z 266.795,A -85,B 0,C 180,E1 -5520.666,E2 -5520.666} C_VEL
LIN {X 0,Y 509.836,Z 266.787,A -85,B 0,C 180,E1 -5523.461,E2 -5523.461} C_VEL
LIN {X 0,Y 509.818,Z 266.789,A -85,B 0,C 180,E1 -5526.352,E2 -5526.352} C_VEL
LIN {X 0,Y 509.839,Z 266.793,A -85,B 0,C 180,E1 -5529.352,E2 -5529.352} C_VEL
LIN {X 0,Y 509.807,Z 266.79,A -85,B 0,C 180,E1 -5532.491,E2 -5532.491} C_VEL
LIN {X 0,Y 509.831,Z 266.794,A -85,B 0,C 180,E1 -5535.329,E2 -5535.329} C_VEL
LIN {X 0,Y 509.848,Z 266.783,A -85,B 0,C 180,E1 -5538.574,E2 -5538.574} C_VEL
LIN {X 0,Y 509.84,Z 266.788,A -85,B 0,C 180,E1 -5541.786,E2 -5541.786} C_VEL
LIN {X 0,Y 509.83,Z 266.785,A -85,B 0,C 180,E1 -5544.622,E2 -5544.622} C_VEL
LIN {X 0,Y 509.85,Z 266.786,A -85,B 0,C 180,E1 -5547.48,E2 -5547.48} C_VEL
LIN {X 0,Y 509.847,Z 266.786,A -85,B 0,C 180,E1 -5550.273,E2 -5550.273} C_VEL
LIN {X 0,Y 509.869,Z 266.777,A -85,B 0,C 180,E1 -5552.944,E2 -5552.944} C_VEL
LIN {X 0,Y 509.838,Z 266.787,A -85,B 0,C 180,E1 -5555.572,E2 -5555.572} C_VEL
LIN {X 0,Y 509.808,Z 266.792,A -85,B 0,C 180,E1 -5558.148,E2 -5558.148} C_VEL
LIN {X 0,Y 509.848,Z 266.786,A -85,B 0,C 180,E1 -5560.681,E2 -5560.681} C_VEL
LIN {X 0,Y 509.864,Z 266.779,A -85,B 0,C 180,E1 -5563.174,E2 -5563.174} C_VEL
LIN {X 0,Y 509.846,Z 266.781,A -85,B 0,C 180,E1 -5565.634,E2 -5565.634} C_VEL
LIN {X 0,Y 509.905,Z 266.778,A -85,B 0,C 180,E1 -5568.874,E2 -5568.874} C_VEL
LIN {X 0,Y 509.937,Z 266.771,A -85,B 0,C 180,E1 -5572.078,E2 -5572.078} C_VEL
LIN {X 0,Y 509.976,Z 266.772,A -85,B 0,C 180,E1 -5574.464,E2 -5574.464} C_VEL
LIN {X 0,Y 510.038,Z 266.757,A -85,B 0,C 180,E1 -5577.631,E2 -5577.631} C_VEL
LIN {X 0,Y 510.037,Z 266.759,A -85,B 0,C 180,E1 -5580,E2 -5580} C_VEL
LIN {X 0,Y 510.038,Z 266.757,A -85,B 0,C 180,E1 -5582.369,E2 -5582.369} C_VEL
LIN {X 0,Y 509.963,Z 266.772,A -85,B 0,C 180,E1 -5585.536,E2 -5585.536} C_VEL
LIN {X 0,Y 509.902,Z 266.776,A -85,B 0,C 180,E1 -5588.721,E2 -5588.721} C_VEL
LIN {X 0,Y 509.891,Z 266.777,A -85,B 0,C 180,E1 -5591.932,E2 -5591.932} C_VEL
LIN {X 0,Y 509.881,Z 266.785,A -85,B 0,C 180,E1 -5595.242,E2 -5595.242} C_VEL
LIN {X 0,Y 509.875,Z 266.784,A -85,B 0,C 180,E1 -5598.001,E2 -5598.001} C_VEL
LIN {X 0,Y 509.838,Z 266.785,A -85,B 0,C 180,E1 -5601.002,E2 -5601.002} C_VEL
LIN {X 0,Y 509.858,Z 266.784,A -85,B 0,C 180,E1 -5604.427,E2 -5604.427} C_VEL
LIN {X 0,Y 509.876,Z 266.779,A -85,B 0,C 180,E1 -5607.056,E2 -5607.056} C_VEL
LIN {X 0,Y 509.87,Z 266.785,A -85,B 0,C 180,E1 -5609.75,E2 -5609.75} C_VEL
LIN {X 0,Y 509.864,Z 266.783,A -85,B 0,C 180,E1 -5612.775,E2 -5612.775} C_VEL
LIN {X 0,Y 509.834,Z 266.785,A -85,B 0,C 180,E1 -5615.582,E2 -5615.582} C_VEL
LIN {X 0,Y 509.844,Z 266.794,A -85,B 0,C 180,E1 -5618.339,E2 -5618.339} C_VEL
LIN {X 0,Y 509.856,Z 266.785,A -85,B 0,C 180,E1 -5621.426,E2 -5621.426} C_VEL
LIN {X 0,Y 509.899,Z 266.93,A -85,B 0,C 180,E1 -5623.928,E2 -5623.928} C_VEL
LIN {X 0,Y 509.801,Z 280.337,A -85,B 0,C 180,E1 -5626.719,E2 -5626.719} C_VEL
LIN {X 0,Y 509.73,Z 295.051,A -85,B 0,C 180,E1 -5629.805,E2 -5629.805} C_VEL
LIN {X 0,Y 511.102,Z 305.599,A -85,B 0,C 180,E1 -5629.996,E2 -5629.996} C_VEL
LIN {X 0,Y 510.998,Z 323.083,A -85,B 0,C 180,E1 -5630.24,E2 -5630.24} C_VEL
LIN {X 0,Y 510.365,Z 328.924,A -85,B 0,C 180,E1 -5630.308,E2 -5630.308} C_VEL
LIN {X 0,Y 504.633,Z 347.891,A -85,B 0,C 180,E1 -5630.444,E2 -5630.444} C_VEL
LIN {X 0,Y 503.942,Z 353.734,A -85,B 0,C 180,E1 -5630.512,E2 -5630.512} C_VEL
LIN {X 0,Y 503.847,Z 373.751,A -85,B 0,C 180,E1 -5630.832,E2 -5630.832} C_VEL
LIN {X 0,Y 503.678,Z 385.851,A -85,B 0,C 180,E1 -5631.198,E2 -5631.198} C_VEL
LIN {X 0,Y 503.488,Z 395.281,A -85,B 0,C 180,E1 -5631.623,E2 -5631.623} C_VEL
LIN {X 0,Y 503.272,Z 404.794,A -85,B 0,C 180,E1 -5632.187,E2 -5632.187} C_VEL
LIN {X 0,Y 503.081,Z 412.683,A -85,B 0,C 180,E1 -5632.777,E2 -5632.777} C_VEL
LIN {X 0,Y 502.836,Z 419.917,A -85,B 0,C 180,E1 -5633.435,E2 -5633.435} C_VEL
LIN {X 0,Y 502.705,Z 426.689,A -85,B 0,C 180,E1 -5634.18,E2 -5634.18} C_VEL
LIN {X 0,Y 502.516,Z 432.951,A -85,B 0,C 180,E1 -5635.013,E2 -5635.013} C_VEL
LIN {X 0,Y 502.368,Z 438.86,A -85,B 0,C 180,E1 -5635.974,E2 -5635.974} C_VEL
LIN {X 0,Y 502.238,Z 444.317,A -85,B 0,C 180,E1 -5637.098,E2 -5637.098} C_VEL
LIN {X 0,Y 502.172,Z 448.52,A -85,B 0,C 180,E1 -5638.28,E2 -5638.28} C_VEL
LIN {X 0,Y 502.112,Z 451.12,A -85,B 0,C 180,E1 -5639.278,E2 -5639.278} C_VEL
LIN {X 0,Y 502.012,Z 453.351,A -85,B 0,C 180,E1 -5640.661,E2 -5640.661} C_VEL
LIN {X 0,Y 501.979,Z 454.118,A -85,B 0,C 180,E1 -5641.889,E2 -5641.889} C_VEL
LIN {X 0,Y 501.995,Z 453.397,A -85,B 0,C 180,E1 -5643.385,E2 -5643.385} C_VEL
LIN {X 0,Y 502.009,Z 452.179,A -85,B 0,C 180,E1 -5644.28,E2 -5644.28} C_VEL
LIN {X 0,Y 502.159,Z 449.483,A -85,B 0,C 180,E1 -5645.466,E2 -5645.466} C_VEL
LIN {X 0,Y 502.21,Z 446.168,A -85,B 0,C 180,E1 -5646.496,E2 -5646.496} C_VEL
LIN {X 0,Y 502.271,Z 442.203,A -85,B 0,C 180,E1 -5647.444,E2 -5647.444} C_VEL
LIN {X 0,Y 502.407,Z 436.848,A -85,B 0,C 180,E1 -5648.458,E2 -5648.458} C_VEL
LIN {X 0,Y 502.567,Z 431.031,A -85,B 0,C 180,E1 -5649.345,E2 -5649.345} C_VEL
LIN {X 0,Y 502.811,Z 422.425,A -85,B 0,C 180,E1 -5650.4,E2 -5650.4} C_VEL
LIN {X 0,Y 503.046,Z 413.312,A -85,B 0,C 180,E1 -5651.257,E2 -5651.257} C_VEL
LIN {X 0,Y 503.292,Z 405.543,A -85,B 0,C 180,E1 -5651.848,E2 -5651.848} C_VEL
LIN {X 0,Y 503.429,Z 397.874,A -85,B 0,C 180,E1 -5652.324,E2 -5652.324} C_VEL
LIN {X 0,Y 503.626,Z 389.161,A -85,B 0,C 180,E1 -5652.751,E2 -5652.751} C_VEL
LIN {X 0,Y 503.739,Z 379.729,A -85,B 0,C 180,E1 -5653.094,E2 -5653.094} C_VEL
LIN {X 0,Y 503.872,Z 369.81,A -85,B 0,C 180,E1 -5653.334,E2 -5653.334} C_VEL
LIN {X 0,Y 504.058,Z 304.163,A -85,B 0,C 180,E1 -5654.288,E2 -5654.288} C_VEL
LIN {X 0,Y 502.662,Z 295.504,A -85,B 0,C 180,E1 -5654.45,E2 -5654.45} C_VEL
LIN {X 0,Y 502.866,Z 282.119,A -85,B 0,C 180,E1 -5657.489,E2 -5657.489} C_VEL
LIN {X 0,Y 503.07,Z 271.407,A -85,B 0,C 180,E1 -5659.943,E2 -5659.943} C_VEL
LIN {X 0,Y 502.931,Z 267.652,A -85,B 0,C 180,E1 -5660.854,E2 -5660.854} C_VEL
LIN {X 0,Y 502.908,Z 267.657,A -85,B 0,C 180,E1 -5663.581,E2 -5663.581} C_VEL
LIN {X 0,Y 502.898,Z 267.648,A -85,B 0,C 180,E1 -5666.796,E2 -5666.796} C_VEL
LIN {X 0,Y 503.035,Z 267.632,A -85,B 0,C 180,E1 -5669.2,E2 -5669.2} C_VEL
LIN {X 0,Y 502.904,Z 267.652,A -85,B 0,C 180,E1 -5671.602,E2 -5671.602} C_VEL
LIN {X 0,Y 502.899,Z 267.648,A -85,B 0,C 180,E1 -5673.204,E2 -5673.204} C_VEL
LIN {X 0,Y 502.888,Z 267.655,A -85,B 0,C 180,E1 -5676.419,E2 -5676.419} C_VEL
LIN {X 0,Y 502.871,Z 267.653,A -85,B 0,C 180,E1 -5678.843,E2 -5678.843} C_VEL
LIN {X 0,Y 502.848,Z 267.66,A -85,B 0,C 180,E1 -5682.101,E2 -5682.101} C_VEL
LIN {X 0,Y 502.85,Z 267.654,A -85,B 0,C 180,E1 -5685.399,E2 -5685.399} C_VEL
LIN {X 0,Y 502.827,Z 267.664,A -85,B 0,C 180,E1 -5688.751,E2 -5688.751} C_VEL
LIN {X 0,Y 502.783,Z 267.664,A -85,B 0,C 180,E1 -5691.31,E2 -5691.31} C_VEL
LIN {X 0,Y 502.783,Z 267.663,A -85,B 0,C 180,E1 -5693.913,E2 -5693.913} C_VEL
LIN {X 0,Y 502.863,Z 267.658,A -85,B 0,C 180,E1 -5696.565,E2 -5696.565} C_VEL
LIN {X 0,Y 502.822,Z 267.662,A -85,B 0,C 180,E1 -5699.287,E2 -5699.287} C_VEL
LIN {X 0,Y 502.779,Z 267.663,A -85,B 0,C 180,E1 -5702.084,E2 -5702.084} C_VEL
LIN {X 0,Y 502.791,Z 267.668,A -85,B 0,C 180,E1 -5704.965,E2 -5704.965} C_VEL
LIN {X 0,Y 502.788,Z 267.663,A -85,B 0,C 180,E1 -5707.953,E2 -5707.953} C_VEL
LIN {X 0,Y 502.814,Z 267.664,A -85,B 0,C 180,E1 -5711.065,E2 -5711.065} C_VEL
LIN {X 0,Y 502.794,Z 267.661,A -85,B 0,C 180,E1 -5714.531,E2 -5714.531} C_VEL
LIN {X 0,Y 502.828,Z 267.663,A -85,B 0,C 180,E1 -5717.864,E2 -5717.864} C_VEL
LIN {X 0,Y 502.802,Z 267.661,A -85,B 0,C 180,E1 -5721.024,E2 -5721.024} C_VEL
LIN {X 0,Y 502.777,Z 267.668,A -85,B 0,C 180,E1 -5724.166,E2 -5724.166} C_VEL
LIN {X 0,Y 502.823,Z 267.658,A -85,B 0,C 180,E1 -5726.992,E2 -5726.992} C_VEL
LIN {X 0,Y 502.821,Z 267.668,A -85,B 0,C 180,E1 -5730.061,E2 -5730.061} C_VEL
LIN {X 0,Y 502.825,Z 267.661,A -85,B 0,C 180,E1 -5732.533,E2 -5732.533} C_VEL
LIN {X 0,Y 502.818,Z 267.658,A -85,B 0,C 180,E1 -5735.298,E2 -5735.298} C_VEL
LIN {X 0,Y 502.769,Z 267.667,A -85,B 0,C 180,E1 -5737.826,E2 -5737.826} C_VEL
LIN {X 0,Y 502.813,Z 267.669,A -85,B 0,C 180,E1 -5740.4,E2 -5740.4} C_VEL
LIN {X 0,Y 502.821,Z 267.661,A -85,B 0,C 180,E1 -5742.931,E2 -5742.931} C_VEL
LIN {X 0,Y 502.832,Z 267.657,A -85,B 0,C 180,E1 -5745.429,E2 -5745.429} C_VEL
LIN {X 0,Y 502.864,Z 267.662,A -85,B 0,C 180,E1 -5748.716,E2 -5748.716} C_VEL
LIN {X 0,Y 502.888,Z 267.65,A -85,B 0,C 180,E1 -5751.966,E2 -5751.966} C_VEL
LIN {X 0,Y 502.92,Z 267.648,A -85,B 0,C 180,E1 -5754.386,E2 -5754.386} C_VEL
LIN {X 0,Y 503.009,Z 267.636,A -85,B 0,C 180,E1 -5757.598,E2 -5757.598} C_VEL
LIN {X 0,Y 503.009,Z 267.634,A -85,B 0,C 180,E1 -5760,E2 -5760} C_VEL
LIN {X 0,Y 503.009,Z 267.635,A -85,B 0,C 180,E1 -5762.402,E2 -5762.402} C_VEL
LIN {X 0,Y 502.929,Z 267.649,A -85,B 0,C 180,E1 -5765.613,E2 -5765.613} C_VEL
LIN {X 0,Y 502.887,Z 267.651,A -85,B 0,C 180,E1 -5768.033,E2 -5768.033} C_VEL
LIN {X 0,Y 502.885,Z 267.656,A -85,B 0,C 180,E1 -5771.283,E2 -5771.283} C_VEL
LIN {X 0,Y 502.831,Z 267.657,A -85,B 0,C 180,E1 -5774.571,E2 -5774.571} C_VEL
LIN {X 0,Y 502.848,Z 267.662,A -85,B 0,C 180,E1 -5777.907,E2 -5777.907} C_VEL
LIN {X 0,Y 502.816,Z 267.659,A -85,B 0,C 180,E1 -5780.537,E2 -5780.537} C_VEL
LIN {X 0,Y 502.782,Z 267.663,A -85,B 0,C 180,E1 -5783.041,E2 -5783.041} C_VEL
LIN {X 0,Y 502.827,Z 267.662,A -85,B 0,C 180,E1 -5785.676,E2 -5785.676} C_VEL
LIN {X 0,Y 502.827,Z 267.663,A -85,B 0,C 180,E1 -5788.373,E2 -5788.373} C_VEL
LIN {X 0,Y 502.781,Z 267.664,A -85,B 0,C 180,E1 -5791.499,E2 -5791.499} C_VEL
LIN {X 0,Y 502.795,Z 267.666,A -85,B 0,C 180,E1 -5793.994,E2 -5793.994} C_VEL
LIN {X 0,Y 502.77,Z 267.665,A -85,B 0,C 180,E1 -5797.179,E2 -5797.179} C_VEL
LIN {X 0,Y 502.777,Z 267.666,A -85,B 0,C 180,E1 -5800.016,E2 -5800.016} C_VEL
LIN {X 0,Y 502.794,Z 267.665,A -85,B 0,C 180,E1 -5802.2,E2 -5802.2} C_VEL
LIN {X 0,Y 502.777,Z 267.664,A -85,B 0,C 180,E1 -5805.471,E2 -5805.471} C_VEL
LIN {X 0,Y 502.787,Z 267.662,A -85,B 0,C 180,E1 -5807.861,E2 -5807.861} C_VEL
LIN {X 0,Y 502.795,Z 267.669,A -85,B 0,C 180,E1 -5811.025,E2 -5811.025} C_VEL
LIN {X 0,Y 502.769,Z 267.665,A -85,B 0,C 180,E1 -5814.17,E2 -5814.17} C_VEL
LIN {X 0,Y 502.825,Z 267.665,A -85,B 0,C 180,E1 -5816.995,E2 -5816.995} C_VEL
LIN {X 0,Y 502.809,Z 267.66,A -85,B 0,C 180,E1 -5820.066,E2 -5820.066} C_VEL
LIN {X 0,Y 502.784,Z 267.664,A -85,B 0,C 180,E1 -5822.531,E2 -5822.531} C_VEL
LIN {X 0,Y 502.768,Z 267.673,A -85,B 0,C 180,E1 -5825.314,E2 -5825.314} C_VEL
LIN {X 0,Y 502.843,Z 267.779,A -85,B 0,C 180,E1 -5827.164,E2 -5827.164} C_VEL
LIN {X 0,Y 503.816,Z 274.421,A -85,B 0,C 180,E1 -5828.521,E2 -5828.521} C_VEL
LIN {X 0,Y 503.379,Z 290.018,A -85,B 0,C 180,E1 -5831.55,E2 -5831.55} C_VEL
LIN {X 0,Y 502.976,Z 306.626,A -85,B 0,C 180,E1 -5834.729,E2 -5834.729} C_VEL
LIN {X 0,Y 502.661,Z 321.599,A -85,B 0,C 180,E1 -5837.563,E2 -5837.563} C_VEL
LIN {X 0,Y 504.132,Z 334.496,A -85,B 0,C 180,E1 -5837.802,E2 -5837.802} C_VEL
LIN {X 0,Y 503.826,Z 398.698,A -85,B 0,C 180,E1 -5838.739,E2 -5838.739} C_VEL
LIN {X 0,Y 503.606,Z 408.498,A -85,B 0,C 180,E1 -5838.988,E2 -5838.988} C_VEL
LIN {X 0,Y 503.463,Z 420.162,A -85,B 0,C 180,E1 -5839.443,E2 -5839.443} C_VEL
LIN {X 0,Y 503.196,Z 430.851,A -85,B 0,C 180,E1 -5840.047,E2 -5840.047} C_VEL
LIN {X 0,Y 502.996,Z 439.206,A -85,B 0,C 180,E1 -5840.652,E2 -5840.652} C_VEL
LIN {X 0,Y 502.794,Z 447.11,A -85,B 0,C 180,E1 -5841.358,E2 -5841.358} C_VEL
LIN {X 0,Y 502.548,Z 454.496,A -85,B 0,C 180,E1 -5842.163,E2 -5842.163} C_VEL
LIN {X 0,Y 502.409,Z 461.994,A -85,B 0,C 180,E1 -5843.172,E2 -5843.172} C_VEL
LIN {X 0,Y 502.316,Z 467.875,A -85,B 0,C 180,E1 -5844.178,E2 -5844.178} C_VEL
LIN {X 0,Y 502.148,Z 472.503,A -85,B 0,C 180,E1 -5845.183,E2 -5845.183} C_VEL
LIN {X 0,Y 502.157,Z 475.511,A -85,B 0,C 180,E1 -5845.987,E2 -5845.987} C_VEL
LIN {X 0,Y 502.133,Z 477.841,A -85,B 0,C 180,E1 -5846.791,E2 -5846.791} C_VEL
LIN {X 0,Y 502.093,Z 479.595,A -85,B 0,C 180,E1 -5847.593,E2 -5847.593} C_VEL
LIN {X 0,Y 502.035,Z 480.85,A -85,B 0,C 180,E1 -5848.396,E2 -5848.396} C_VEL
LIN {X 0,Y 501.988,Z 481.631,A -85,B 0,C 180,E1 -5849.198,E2 -5849.198} C_VEL
LIN {X 0,Y 501.98,Z 481.924,A -85,B 0,C 180,E1 -5850,E2 -5850} C_VEL
LIN {X 0,Y 501.988,Z 481.625,A -85,B 0,C 180,E1 -5850.802,E2 -5850.802} C_VEL
LIN {X 0,Y 502.035,Z 480.841,A -85,B 0,C 180,E1 -5851.604,E2 -5851.604} C_VEL
LIN {X 0,Y 502.093,Z 479.582,A -85,B 0,C 180,E1 -5852.407,E2 -5852.407} C_VEL
LIN {X 0,Y 502.166,Z 476.665,A -85,B 0,C 180,E1 -5853.611,E2 -5853.611} C_VEL
LIN {X 0,Y 502.137,Z 474.005,A -85,B 0,C 180,E1 -5854.415,E2 -5854.415} C_VEL
LIN {X 0,Y 502.272,Z 468.804,A -85,B 0,C 180,E1 -5855.621,E2 -5855.621} C_VEL
LIN {X 0,Y 502.365,Z 463.087,A -85,B 0,C 180,E1 -5856.648,E2 -5856.648} C_VEL
LIN {X 0,Y 502.502,Z 456.158,A -85,B 0,C 180,E1 -5857.635,E2 -5857.635} C_VEL
LIN {X 0,Y 502.746,Z 448.089,A -85,B 0,C 180,E1 -5858.541,E2 -5858.541} C_VEL
LIN {X 0,Y 502.959,Z 440.385,A -85,B 0,C 180,E1 -5859.247,E2 -5859.247} C_VEL
LIN {X 0,Y 503.141,Z 432.29,A -85,B 0,C 180,E1 -5859.852,E2 -5859.852} C_VEL
LIN {X 0,Y 503.338,Z 423.898,A -85,B 0,C 180,E1 -5860.356,E2 -5860.356} C_VEL
LIN {X 0,Y 503.513,Z 415.323,A -85,B 0,C 180,E1 -5860.759,E2 -5860.759} C_VEL
LIN {X 0,Y 503.649,Z 405.918,A -85,B 0,C 180,E1 -5861.087,E2 -5861.087} C_VEL
LIN {X 0,Y 503.916,Z 394.024,A -85,B 0,C 180,E1 -5861.347,E2 -5861.347} C_VEL
LIN {X 0,Y 504.034,Z 332.299,A -85,B 0,C 180,E1 -5862.23,E2 -5862.23} C_VEL
LIN {X 0,Y 502.63,Z 321.393,A -85,B 0,C 180,E1 -5862.445,E2 -5862.445} C_VEL
LIN {X 0,Y 502.936,Z 305.63,A -85,B 0,C 180,E1 -5865.396,E2 -5865.396} C_VEL
LIN {X 0,Y 503.295,Z 289.477,A -85,B 0,C 180,E1 -5868.442,E2 -5868.442} C_VEL
LIN {X 0,Y 503.656,Z 274.636,A -85,B 0,C 180,E1 -5871.272,E2 -5871.272} C_VEL
LIN {X 0,Y 503.053,Z 268.766,A -85,B 0,C 180,E1 -5872.431,E2 -5872.431} C_VEL
LIN {X 0,Y 502.828,Z 267.667,A -85,B 0,C 180,E1 -5872.667,E2 -5872.667} C_VEL
LIN {X 0,Y 502.776,Z 267.667,A -85,B 0,C 180,E1 -5875.678,E2 -5875.678} C_VEL
LIN {X 0,Y 502.77,Z 267.671,A -85,B 0,C 180,E1 -5878.376,E2 -5878.376} C_VEL
LIN {X 0,Y 502.787,Z 267.667,A -85,B 0,C 180,E1 -5881.143,E2 -5881.143} C_VEL
LIN {X 0,Y 502.783,Z 267.664,A -85,B 0,C 180,E1 -5883.994,E2 -5883.994} C_VEL
LIN {X 0,Y 502.771,Z 267.674,A -85,B 0,C 180,E1 -5887.177,E2 -5887.177} C_VEL
LIN {X 0,Y 502.779,Z 267.666,A -85,B 0,C 180,E1 -5890.015,E2 -5890.015} C_VEL
LIN {X 0,Y 502.796,Z 267.662,A -85,B 0,C 180,E1 -5892.198,E2 -5892.198} C_VEL
LIN {X 0,Y 502.778,Z 267.673,A -85,B 0,C 180,E1 -5895.469,E2 -5895.469} C_VEL
LIN {X 0,Y 502.811,Z 267.661,A -85,B 0,C 180,E1 -5898.933,E2 -5898.933} C_VEL
LIN {X 0,Y 502.783,Z 267.664,A -85,B 0,C 180,E1 -5902.045,E2 -5902.045} C_VEL
LIN {X 0,Y 502.795,Z 267.663,A -85,B 0,C 180,E1 -5905.034,E2 -5905.034} C_VEL
LIN {X 0,Y 502.772,Z 267.671,A -85,B 0,C 180,E1 -5907.915,E2 -5907.915} C_VEL
LIN {X 0,Y 502.811,Z 267.659,A -85,B 0,C 180,E1 -5910.711,E2 -5910.711} C_VEL
LIN {X 0,Y 502.851,Z 267.653,A -85,B 0,C 180,E1 -5913.439,E2 -5913.439} C_VEL
LIN {X 0,Y 502.763,Z 267.674,A -85,B 0,C 180,E1 -5916.085,E2 -5916.085} C_VEL
LIN {X 0,Y 502.77,Z 267.664,A -85,B 0,C 180,E1 -5918.688,E2 -5918.688} C_VEL
LIN {X 0,Y 502.815,Z 267.659,A -85,B 0,C 180,E1 -5921.248,E2 -5921.248} C_VEL
LIN {X 0,Y 502.805,Z 267.66,A -85,B 0,C 180,E1 -5923.767,E2 -5923.767} C_VEL
LIN {X 0,Y 502.813,Z 267.663,A -85,B 0,C 180,E1 -5926.254,E2 -5926.254} C_VEL
LIN {X 0,Y 502.868,Z 267.657,A -85,B 0,C 180,E1 -5928.717,E2 -5928.717} C_VEL
LIN {X 0,Y 502.887,Z 267.648,A -85,B 0,C 180,E1 -5931.967,E2 -5931.967} C_VEL
LIN {X 0,Y 502.928,Z 267.649,A -85,B 0,C 180,E1 -5934.386,E2 -5934.386} C_VEL
LIN {X 0,Y 503.009,Z 267.633,A -85,B 0,C 180,E1 -5937.598,E2 -5937.598} C_VEL
LIN {X 0,Y 503.009,Z 267.634,A -85,B 0,C 180,E1 -5940,E2 -5940} C_VEL
LIN {X 0,Y 503.008,Z 267.632,A -85,B 0,C 180,E1 -5942.402,E2 -5942.402} C_VEL
LIN {X 0,Y 502.916,Z 267.649,A -85,B 0,C 180,E1 -5945.614,E2 -5945.614} C_VEL
LIN {X 0,Y 502.86,Z 267.654,A -85,B 0,C 180,E1 -5948.844,E2 -5948.844} C_VEL
LIN {X 0,Y 502.832,Z 267.655,A -85,B 0,C 180,E1 -5952.102,E2 -5952.102} C_VEL
LIN {X 0,Y 502.835,Z 267.665,A -85,B 0,C 180,E1 -5955.4,E2 -5955.4} C_VEL
LIN {X 0,Y 502.833,Z 267.66,A -85,B 0,C 180,E1 -5958.123,E2 -5958.123} C_VEL
LIN {X 0,Y 502.816,Z 267.659,A -85,B 0,C 180,E1 -5960.537,E2 -5960.537} C_VEL
LIN {X 0,Y 502.782,Z 267.665,A -85,B 0,C 180,E1 -5963.041,E2 -5963.041} C_VEL
LIN {X 0,Y 502.83,Z 267.665,A -85,B 0,C 180,E1 -5965.676,E2 -5965.676} C_VEL
LIN {X 0,Y 502.831,Z 267.66,A -85,B 0,C 180,E1 -5968.373,E2 -5968.373} C_VEL
LIN {X 0,Y 502.784,Z 267.665,A -85,B 0,C 180,E1 -5971.5,E2 -5971.5} C_VEL
LIN {X 0,Y 502.797,Z 267.666,A -85,B 0,C 180,E1 -5974.446,E2 -5974.446} C_VEL
LIN {X 0,Y 502.773,Z 267.666,A -85,B 0,C 180,E1 -5977.179,E2 -5977.179} C_VEL
LIN {X 0,Y 502.814,Z 267.665,A -85,B 0,C 180,E1 -5980.013,E2 -5980.013} C_VEL
LIN {X 0,Y 502.851,Z 267.658,A -85,B 0,C 180,E1 -5983.386,E2 -5983.386} C_VEL
LIN {X 0,Y 502.862,Z 267.848,A -85,B 0,C 180,E1 -5983.884,E2 -5983.884} C_VEL
LIN {X 0,Y 502.761,Z 280.923,A -85,B 0,C 180,E1 -5986.627,E2 -5986.627} C_VEL
LIN {X 0,Y 502.684,Z 295.155,A -85,B 0,C 180,E1 -5989.625,E2 -5989.625} C_VEL
LIN {X 0,Y 504.188,Z 306.377,A -85,B 0,C 180,E1 -5989.836,E2 -5989.836} C_VEL
LIN {X 0,Y 503.942,Z 353.734,A -85,B 0,C 180,E1 -5990.512,E2 -5990.512} C_VEL
LIN {X 0,Y 503.274,Z 359.583,A -85,B 0,C 180,E1 -5990.578,E2 -5990.578} C_VEL
LIN {X 0,Y 500.445,Z 369.07,A -85,B 0,C 180,E1 -5990.66,E2 -5990.66} C_VEL
LIN {X 0,Y 497.516,Z 378.446,A -85,B 0,C 180,E1 -5990.801,E2 -5990.801} C_VEL
LIN {X 0,Y 496.746,Z 384.109,A -85,B 0,C 180,E1 -5990.969,E2 -5990.969} C_VEL
LIN {X 0,Y 496.506,Z 395.566,A -85,B 0,C 180,E1 -5991.479,E2 -5991.479} C_VEL
LIN {X 0,Y 496.307,Z 403.974,A -85,B 0,C 180,E1 -5991.978,E2 -5991.978} C_VEL
LIN {X 0,Y 496.106,Z 411.917,A -85,B 0,C 180,E1 -5992.565,E2 -5992.565} C_VEL
LIN {X 0,Y 495.857,Z 419.147,A -85,B 0,C 180,E1 -5993.215,E2 -5993.215} C_VEL
LIN {X 0,Y 495.685,Z 425.636,A -85,B 0,C 180,E1 -5993.917,E2 -5993.917} C_VEL
LIN {X 0,Y 495.536,Z 431.643,A -85,B 0,C 180,E1 -5994.696,E2 -5994.696} C_VEL
LIN {X 0,Y 495.369,Z 436.413,A -85,B 0,C 180,E1 -5995.425,E2 -5995.425} C_VEL
LIN {X 0,Y 495.261,Z 441.626,A -85,B 0,C 180,E1 -5996.399,E2 -5996.399} C_VEL
LIN {X 0,Y 495.127,Z 445.754,A -85,B 0,C 180,E1 -5997.359,E2 -5997.359} C_VEL
LIN {X 0,Y 495.092,Z 449.202,A -85,B 0,C 180,E1 -5998.4,E2 -5998.4} C_VEL
LIN {X 0,Y 495.031,Z 451.367,A -85,B 0,C 180,E1 -5999.264,E2 -5999.264} C_VEL
LIN {X 0,Y 494.934,Z 453.028,A -85,B 0,C 180,E1 -6000.2,E2 -6000.2} C_VEL
LIN {X 0,Y 494.912,Z 454.02,A -85,B 0,C 180,E1 -6001.131,E2 -6001.131} C_VEL
LIN {X 0,Y 494.906,Z 454.35,A -85,B 0,C 180,E1 -6002.056,E2 -6002.056} C_VEL
LIN {X 0,Y 494.9,Z 453.521,A -85,B 0,C 180,E1 -6003.464,E2 -6003.464} C_VEL
LIN {X 0,Y 494.979,Z 451.423,A -85,B 0,C 180,E1 -6004.79,E2 -6004.79} C_VEL
LIN {X 0,Y 495.127,Z 447.89,A -85,B 0,C 180,E1 -6006.139,E2 -6006.139} C_VEL
LIN {X 0,Y 495.185,Z 443.433,A -85,B 0,C 180,E1 -6007.298,E2 -6007.298} C_VEL
LIN {X 0,Y 495.329,Z 438.158,A -85,B 0,C 180,E1 -6008.353,E2 -6008.353} C_VEL
LIN {X 0,Y 495.482,Z 432.725,A -85,B 0,C 180,E1 -6009.232,E2 -6009.232} C_VEL
LIN {X 0,Y 495.622,Z 427.771,A -85,B 0,C 180,E1 -6009.908,E2 -6009.908} C_VEL
LIN {X 0,Y 495.843,Z 420.213,A -85,B 0,C 180,E1 -6010.76,E2 -6010.76} C_VEL
LIN {X 0,Y 496.024,Z 413.85,A -85,B 0,C 180,E1 -6011.358,E2 -6011.358} C_VEL
LIN {X 0,Y 496.289,Z 406.172,A -85,B 0,C 180,E1 -6011.955,E2 -6011.955} C_VEL
LIN {X 0,Y 496.478,Z 397.576,A -85,B 0,C 180,E1 -6012.494,E2 -6012.494} C_VEL
LIN {X 0,Y 496.645,Z 388.777,A -85,B 0,C 180,E1 -6012.925,E2 -6012.925} C_VEL
LIN {X 0,Y 496.823,Z 379.026,A -85,B 0,C 180,E1 -6013.275,E2 -6013.275} C_VEL
LIN {X 0,Y 496.935,Z 368.688,A -85,B 0,C 180,E1 -6013.517,E2 -6013.517} C_VEL
LIN {X 0,Y 497.177,Z 305.286,A -85,B 0,C 180,E1 -6014.445,E2 -6014.445} C_VEL
LIN {X 0,Y 495.632,Z 295.644,A -85,B 0,C 180,E1 -6014.63,E2 -6014.63} C_VEL
LIN {X 0,Y 495.886,Z 281.263,A -85,B 0,C 180,E1 -6017.935,E2 -6017.935} C_VEL
LIN {X 0,Y 496.058,Z 271.438,A -85,B 0,C 180,E1 -6020.212,E2 -6020.212} C_VEL
LIN {X 0,Y 495.88,Z 268.531,A -85,B 0,C 180,E1 -6020.929,E2 -6020.929} C_VEL
LIN {X 0,Y 495.862,Z 268.534,A -85,B 0,C 180,E1 -6023.49,E2 -6023.49} C_VEL
LIN {X 0,Y 495.842,Z 268.527,A -85,B 0,C 180,E1 -6026.75,E2 -6026.75} C_VEL
LIN {X 0,Y 495.871,Z 268.526,A -85,B 0,C 180,E1 -6028.376,E2 -6028.376} C_VEL
LIN {X 0,Y 495.985,Z 268.51,A -85,B 0,C 180,E1 -6030.812,E2 -6030.812} C_VEL
LIN {X 0,Y 495.995,Z 268.511,A -85,B 0,C 180,E1 -6032.436,E2 -6032.436} C_VEL
LIN {X 0,Y 495.883,Z 268.526,A -85,B 0,C 180,E1 -6035.693,E2 -6035.693} C_VEL
LIN {X 0,Y 495.84,Z 268.528,A -85,B 0,C 180,E1 -6038.969,E2 -6038.969} C_VEL
LIN {X 0,Y 495.83,Z 268.534,A -85,B 0,C 180,E1 -6042.034,E2 -6042.034} C_VEL
LIN {X 0,Y 495.825,Z 268.529,A -85,B 0,C 180,E1 -6045.451,E2 -6045.451} C_VEL
LIN {X 0,Y 495.779,Z 268.54,A -85,B 0,C 180,E1 -6048.237,E2 -6048.237} C_VEL
LIN {X 0,Y 495.774,Z 268.544,A -85,B 0,C 180,E1 -6050.756,E2 -6050.756} C_VEL
LIN {X 0,Y 495.746,Z 268.54,A -85,B 0,C 180,E1 -6053.387,E2 -6053.387} C_VEL
LIN {X 0,Y 495.788,Z 268.534,A -85,B 0,C 180,E1 -6056.067,E2 -6056.067} C_VEL
LIN {X 0,Y 495.771,Z 268.544,A -85,B 0,C 180,E1 -6058.814,E2 -6058.814} C_VEL
LIN {X 0,Y 495.752,Z 268.539,A -85,B 0,C 180,E1 -6061.724,E2 -6061.724} C_VEL
LIN {X 0,Y 495.759,Z 268.541,A -85,B 0,C 180,E1 -6064.692,E2 -6064.692} C_VEL
LIN {X 0,Y 495.724,Z 268.547,A -85,B 0,C 180,E1 -6067.561,E2 -6067.561} C_VEL
LIN {X 0,Y 495.761,Z 268.539,A -85,B 0,C 180,E1 -6070.699,E2 -6070.699} C_VEL
LIN {X 0,Y 495.728,Z 268.544,A -85,B 0,C 180,E1 -6074,E2 -6074} C_VEL
LIN {X 0,Y 495.756,Z 268.541,A -85,B 0,C 180,E1 -6077.12,E2 -6077.12} C_VEL
LIN {X 0,Y 495.775,Z 268.537,A -85,B 0,C 180,E1 -6080.364,E2 -6080.364} C_VEL
LIN {X 0,Y 495.725,Z 268.546,A -85,B 0,C 180,E1 -6083.456,E2 -6083.456} C_VEL
LIN {X 0,Y 495.752,Z 268.541,A -85,B 0,C 180,E1 -6086.435,E2 -6086.435} C_VEL
LIN {X 0,Y 495.747,Z 268.54,A -85,B 0,C 180,E1 -6089.312,E2 -6089.312} C_VEL
LIN {X 0,Y 495.773,Z 268.546,A -85,B 0,C 180,E1 -6092.108,E2 -6092.108} C_VEL
LIN {X 0,Y 495.778,Z 268.537,A -85,B 0,C 180,E1 -6094.832,E2 -6094.832} C_VEL
LIN {X 0,Y 495.738,Z 268.541,A -85,B 0,C 180,E1 -6097.494,E2 -6097.494} C_VEL
LIN {X 0,Y 495.76,Z 268.543,A -85,B 0,C 180,E1 -6100.109,E2 -6100.109} C_VEL
LIN {X 0,Y 495.774,Z 268.542,A -85,B 0,C 180,E1 -6102.681,E2 -6102.681} C_VEL
LIN {X 0,Y 495.777,Z 268.537,A -85,B 0,C 180,E1 -6105.217,E2 -6105.217} C_VEL
LIN {X 0,Y 495.838,Z 268.535,A -85,B 0,C 180,E1 -6108.554,E2 -6108.554} C_VEL
LIN {X 0,Y 495.86,Z 268.525,A -85,B 0,C 180,E1 -6111.852,E2 -6111.852} C_VEL
LIN {X 0,Y 495.876,Z 268.525,A -85,B 0,C 180,E1 -6114.306,E2 -6114.306} C_VEL
LIN {X 0,Y 495.978,Z 268.512,A -85,B 0,C 180,E1 -6117.564,E2 -6117.564} C_VEL
LIN {X 0,Y 495.981,Z 268.51,A -85,B 0,C 180,E1 -6120,E2 -6120} C_VEL
LIN {X 0,Y 495.978,Z 268.511,A -85,B 0,C 180,E1 -6122.436,E2 -6122.436} C_VEL
LIN {X 0,Y 495.884,Z 268.526,A -85,B 0,C 180,E1 -6125.694,E2 -6125.694} C_VEL
LIN {X 0,Y 495.859,Z 268.526,A -85,B 0,C 180,E1 -6128.148,E2 -6128.148} C_VEL
LIN {X 0,Y 495.859,Z 268.534,A -85,B 0,C 180,E1 -6131.445,E2 -6131.445} C_VEL
LIN {X 0,Y 495.776,Z 268.536,A -85,B 0,C 180,E1 -6134.783,E2 -6134.783} C_VEL
LIN {X 0,Y 495.772,Z 268.54,A -85,B 0,C 180,E1 -6137.319,E2 -6137.319} C_VEL
LIN {X 0,Y 495.759,Z 268.546,A -85,B 0,C 180,E1 -6139.891,E2 -6139.891} C_VEL
LIN {X 0,Y 495.749,Z 268.539,A -85,B 0,C 180,E1 -6142.862,E2 -6142.862} C_VEL
LIN {X 0,Y 495.779,Z 268.544,A -85,B 0,C 180,E1 -6146.068,E2 -6146.068} C_VEL
LIN {X 0,Y 495.759,Z 268.539,A -85,B 0,C 180,E1 -6148.816,E2 -6148.816} C_VEL
LIN {X 0,Y 495.744,Z 268.542,A -85,B 0,C 180,E1 -6151.726,E2 -6151.726} C_VEL
LIN {X 0,Y 495.764,Z 268.541,A -85,B 0,C 180,E1 -6154.695,E2 -6154.695} C_VEL
LIN {X 0,Y 495.72,Z 268.543,A -85,B 0,C 180,E1 -6157.562,E2 -6157.562} C_VEL
LIN {X 0,Y 495.757,Z 268.545,A -85,B 0,C 180,E1 -6160.701,E2 -6160.701} C_VEL
LIN {X 0,Y 495.719,Z 268.544,A -85,B 0,C 180,E1 -6164.002,E2 -6164.002} C_VEL
LIN {X 0,Y 495.709,Z 268.548,A -85,B 0,C 180,E1 -6167.117,E2 -6167.117} C_VEL
LIN {X 0,Y 495.749,Z 268.541,A -85,B 0,C 180,E1 -6170.363,E2 -6170.363} C_VEL
LIN {X 0,Y 495.722,Z 268.545,A -85,B 0,C 180,E1 -6173.457,E2 -6173.457} C_VEL
LIN {X 0,Y 495.746,Z 268.54,A -85,B 0,C 180,E1 -6176.436,E2 -6176.436} C_VEL
LIN {X 0,Y 495.745,Z 268.547,A -85,B 0,C 180,E1 -6179.313,E2 -6179.313} C_VEL
LIN {X 0,Y 495.731,Z 268.543,A -85,B 0,C 180,E1 -6182.107,E2 -6182.107} C_VEL
LIN {X 0,Y 495.726,Z 268.549,A -85,B 0,C 180,E1 -6185.14,E2 -6185.14} C_VEL
LIN {X 0,Y 495.787,Z 268.544,A -85,B 0,C 180,E1 -6187.011,E2 -6187.011} C_VEL
LIN {X 0,Y 496.826,Z 275.336,A -85,B 0,C 180,E1 -6188.421,E2 -6188.421} C_VEL
LIN {X 0,Y 496.386,Z 290.159,A -85,B 0,C 180,E1 -6191.343,E2 -6191.343} C_VEL
LIN {X 0,Y 495.965,Z 306.349,A -85,B 0,C 180,E1 -6194.49,E2 -6194.49} C_VEL
LIN {X 0,Y 495.625,Z 321.566,A -85,B 0,C 180,E1 -6197.404,E2 -6197.404} C_VEL
LIN {X 0,Y 497.201,Z 335.352,A -85,B 0,C 180,E1 -6197.645,E2 -6197.645} C_VEL
LIN {X 0,Y 496.878,Z 398.405,A -85,B 0,C 180,E1 -6198.579,E2 -6198.579} C_VEL
LIN {X 0,Y 496.647,Z 408.24,A -85,B 0,C 180,E1 -6198.832,E2 -6198.832} C_VEL
LIN {X 0,Y 496.485,Z 419.931,A -85,B 0,C 180,E1 -6199.293,E2 -6199.293} C_VEL
LIN {X 0,Y 496.183,Z 430.632,A -85,B 0,C 180,E1 -6199.905,E2 -6199.905} C_VEL
LIN {X 0,Y 495.983,Z 438.994,A -85,B 0,C 180,E1 -6200.519,E2 -6200.519} C_VEL
LIN {X 0,Y 495.756,Z 446.902,A -85,B 0,C 180,E1 -6201.234,E2 -6201.234} C_VEL
LIN {X 0,Y 495.493,Z 454.29,A -85,B 0,C 180,E1 -6202.051,E2 -6202.051} C_VEL
LIN {X 0,Y 495.339,Z 462.06,A -85,B 0,C 180,E1 -6203.114,E2 -6203.114} C_VEL
LIN {X 0,Y 495.202,Z 468.638,A -85,B 0,C 180,E1 -6204.299,E2 -6204.299} C_VEL
LIN {X 0,Y 495.041,Z 473.829,A -85,B 0,C 180,E1 -6205.522,E2 -6205.522} C_VEL
LIN {X 0,Y 495.086,Z 476.488,A -85,B 0,C 180,E1 -6206.338,E2 -6206.338} C_VEL
LIN {X 0,Y 495,Z 479.398,A -85,B 0,C 180,E1 -6207.559,E2 -6207.559} C_VEL
LIN {X 0,Y 494.961,Z 480.655,A -85,B 0,C 180,E1 -6208.373,E2 -6208.373} C_VEL
LIN {X 0,Y 494.908,Z 481.435,A -85,B 0,C 180,E1 -6209.186,E2 -6209.186} C_VEL
LIN {X 0,Y 494.897,Z 481.728,A -85,B 0,C 180,E1 -6210,E2 -6210} C_VEL
LIN {X 0,Y 494.908,Z 481.429,A -85,B 0,C 180,E1 -6210.814,E2 -6210.814} C_VEL
LIN {X 0,Y 494.961,Z 480.644,A -85,B 0,C 180,E1 -6211.627,E2 -6211.627} C_VEL
LIN {X 0,Y 495,Z 479.383,A -85,B 0,C 180,E1 -6212.441,E2 -6212.441} C_VEL
LIN {X 0,Y 495.087,Z 476.465,A -85,B 0,C 180,E1 -6213.662,E2 -6213.662} C_VEL
LIN {X 0,Y 495.042,Z 473.802,A -85,B 0,C 180,E1 -6214.478,E2 -6214.478} C_VEL
LIN {X 0,Y 495.202,Z 468.599,A -85,B 0,C 180,E1 -6215.701,E2 -6215.701} C_VEL
LIN {X 0,Y 495.337,Z 462.009,A -85,B 0,C 180,E1 -6216.886,E2 -6216.886} C_VEL
LIN {X 0,Y 495.493,Z 454.241,A -85,B 0,C 180,E1 -6217.949,E2 -6217.949} C_VEL
LIN {X 0,Y 495.756,Z 446.851,A -85,B 0,C 180,E1 -6218.765,E2 -6218.765} C_VEL
LIN {X 0,Y 495.982,Z 438.936,A -85,B 0,C 180,E1 -6219.481,E2 -6219.481} C_VEL
LIN {X 0,Y 496.178,Z 430.57,A -85,B 0,C 180,E1 -6220.095,E2 -6220.095} C_VEL
LIN {X 0,Y 496.456,Z 419.871,A -85,B 0,C 180,E1 -6220.708,E2 -6220.708} C_VEL
LIN {X 0,Y 496.623,Z 409.022,A -85,B 0,C 180,E1 -6221.143,E2 -6221.143} C_VEL
LIN {X 0,Y 496.848,Z 399.663,A -85,B 0,C 180,E1 -6221.396,E2 -6221.396} C_VEL
LIN {X 0,Y 497.057,Z 372.215,A -85,B 0,C 180,E1 -6221.82,E2 -6221.82} C_VEL
LIN {X 0,Y 496.977,Z 332.119,A -85,B 0,C 180,E1 -6222.407,E2 -6222.407} C_VEL
LIN {X 0,Y 495.602,Z 321.223,A -85,B 0,C 180,E1 -6222.618,E2 -6222.618} C_VEL
LIN {X 0,Y 495.964,Z 304.297,A -85,B 0,C 180,E1 -6225.829,E2 -6225.829} C_VEL
LIN {X 0,Y 496.293,Z 289.591,A -85,B 0,C 180,E1 -6228.644,E2 -6228.644} C_VEL
LIN {X 0,Y 496.662,Z 276.376,A -85,B 0,C 180,E1 -6231.2,E2 -6231.2} C_VEL
LIN {X 0,Y 496.235,Z 271.056,A -85,B 0,C 180,E1 -6232.262,E2 -6232.262} C_VEL
LIN {X 0,Y 495.8,Z 268.542,A -85,B 0,C 180,E1 -6232.777,E2 -6232.777} C_VEL
LIN {X 0,Y 495.719,Z 268.548,A -85,B 0,C 180,E1 -6236.071,E2 -6236.071} C_VEL
LIN {X 0,Y 495.724,Z 268.551,A -85,B 0,C 180,E1 -6238.817,E2 -6238.817} C_VEL
LIN {X 0,Y 495.749,Z 268.54,A -85,B 0,C 180,E1 -6241.724,E2 -6241.724} C_VEL
LIN {X 0,Y 495.757,Z 268.545,A -85,B 0,C 180,E1 -6244.692,E2 -6244.692} C_VEL
LIN {X 0,Y 495.722,Z 268.548,A -85,B 0,C 180,E1 -6247.561,E2 -6247.561} C_VEL
LIN {X 0,Y 495.75,Z 268.542,A -85,B 0,C 180,E1 -6250.046,E2 -6250.046} C_VEL
LIN {X 0,Y 495.709,Z 268.549,A -85,B 0,C 180,E1 -6252.883,E2 -6252.883} C_VEL
LIN {X 0,Y 495.719,Z 268.546,A -85,B 0,C 180,E1 -6255.997,E2 -6255.997} C_VEL
LIN {X 0,Y 495.757,Z 268.544,A -85,B 0,C 180,E1 -6259.299,E2 -6259.299} C_VEL
LIN {X 0,Y 495.72,Z 268.541,A -85,B 0,C 180,E1 -6262.438,E2 -6262.438} C_VEL
LIN {X 0,Y 495.77,Z 268.543,A -85,B 0,C 180,E1 -6265.456,E2 -6265.456} C_VEL
LIN {X 0,Y 495.744,Z 268.541,A -85,B 0,C 180,E1 -6268.363,E2 -6268.363} C_VEL
LIN {X 0,Y 495.775,Z 268.539,A -85,B 0,C 180,E1 -6271.507,E2 -6271.507} C_VEL
LIN {X 0,Y 495.768,Z 268.542,A -85,B 0,C 180,E1 -6273.931,E2 -6273.931} C_VEL
LIN {X 0,Y 495.746,Z 268.538,A -85,B 0,C 180,E1 -6277.139,E2 -6277.139} C_VEL
LIN {X 0,Y 495.757,Z 268.543,A -85,B 0,C 180,E1 -6280.109,E2 -6280.109} C_VEL
LIN {X 0,Y 495.766,Z 268.539,A -85,B 0,C 180,E1 -6282.681,E2 -6282.681} C_VEL
LIN {X 0,Y 495.774,Z 268.534,A -85,B 0,C 180,E1 -6285.217,E2 -6285.217} C_VEL
LIN {X 0,Y 495.842,Z 268.535,A -85,B 0,C 180,E1 -6288.555,E2 -6288.555} C_VEL
LIN {X 0,Y 495.859,Z 268.523,A -85,B 0,C 180,E1 -6291.852,E2 -6291.852} C_VEL
LIN {X 0,Y 495.883,Z 268.525,A -85,B 0,C 180,E1 -6294.306,E2 -6294.306} C_VEL
LIN {X 0,Y 495.978,Z 268.509,A -85,B 0,C 180,E1 -6297.564,E2 -6297.564} C_VEL
LIN {X 0,Y 495.98,Z 268.51,A -85,B 0,C 180,E1 -6300,E2 -6300} C_VEL
LIN {X 0,Y 495.977,Z 268.508,A -85,B 0,C 180,E1 -6302.436,E2 -6302.436} C_VEL
LIN {X 0,Y 495.871,Z 268.525,A -85,B 0,C 180,E1 -6305.694,E2 -6305.694} C_VEL
LIN {X 0,Y 495.829,Z 268.532,A -85,B 0,C 180,E1 -6308.97,E2 -6308.97} C_VEL
LIN {X 0,Y 495.815,Z 268.529,A -85,B 0,C 180,E1 -6312.035,E2 -6312.035} C_VEL
LIN {X 0,Y 495.811,Z 268.541,A -85,B 0,C 180,E1 -6315.452,E2 -6315.452} C_VEL
LIN {X 0,Y 495.794,Z 268.536,A -85,B 0,C 180,E1 -6318.248,E2 -6318.248} C_VEL
LIN {X 0,Y 495.762,Z 268.537,A -85,B 0,C 180,E1 -6320.757,E2 -6320.757} C_VEL
LIN {X 0,Y 495.74,Z 268.546,A -85,B 0,C 180,E1 -6323.388,E2 -6323.388} C_VEL
LIN {X 0,Y 495.789,Z 268.541,A -85,B 0,C 180,E1 -6326.068,E2 -6326.068} C_VEL
LIN {X 0,Y 495.768,Z 268.537,A -85,B 0,C 180,E1 -6328.815,E2 -6328.815} C_VEL
LIN {X 0,Y 495.746,Z 268.544,A -85,B 0,C 180,E1 -6331.726,E2 -6331.726} C_VEL
LIN {X 0,Y 495.767,Z 268.539,A -85,B 0,C 180,E1 -6334.696,E2 -6334.696} C_VEL
LIN {X 0,Y 495.724,Z 268.545,A -85,B 0,C 180,E1 -6337.562,E2 -6337.562} C_VEL
LIN {X 0,Y 495.772,Z 268.545,A -85,B 0,C 180,E1 -6340.7,E2 -6340.7} C_VEL
LIN {X 0,Y 495.831,Z 268.698,A -85,B 0,C 180,E1 -6343.814,E2 -6343.814} C_VEL
LIN {X 0,Y 495.78,Z 280.485,A -85,B 0,C 180,E1 -6346.299,E2 -6346.299} C_VEL
LIN {X 0,Y 495.693,Z 295.58,A -85,B 0,C 180,E1 -6349.46,E2 -6349.46} C_VEL
LIN {X 0,Y 497.246,Z 306.204,A -85,B 0,C 180,E1 -6349.656,E2 -6349.656} C_VEL
LIN {X 0,Y 496.878,Z 371.799,A -85,B 0,C 180,E1 -6350.63,E2 -6350.63} C_VEL
LIN {X 0,Y 496.774,Z 381.715,A -85,B 0,C 180,E1 -6350.893,E2 -6350.893} C_VEL
LIN {X 0,Y 496.746,Z 384.109,A -85,B 0,C 180,E1 -6350.969,E2 -6350.969} C_VEL
LIN {X 0,Y 495.967,Z 387.889,A -85,B 0,C 180,E1 -6351.096,E2 -6351.096} C_VEL
LIN {X 0,Y 493.002,Z 393.77,A -85,B 0,C 180,E1 -6351.288,E2 -6351.288} C_VEL
LIN {X 0,Y 490.074,Z 399.459,A -85,B 0,C 180,E1 -6351.536,E2 -6351.536} C_VEL
LIN {X 0,Y 489.344,Z 402.926,A -85,B 0,C 180,E1 -6351.746,E2 -6351.746} C_VEL
LIN {X 0,Y 489.104,Z 411.888,A -85,B 0,C 180,E1 -6352.409,E2 -6352.409} C_VEL
LIN {X 0,Y 488.857,Z 419.248,A -85,B 0,C 180,E1 -6353.078,E2 -6353.078} C_VEL
LIN {X 0,Y 488.653,Z 426.385,A -85,B 0,C 180,E1 -6353.867,E2 -6353.867} C_VEL
LIN {X 0,Y 488.493,Z 432.021,A -85,B 0,C 180,E1 -6354.615,E2 -6354.615} C_VEL
LIN {X 0,Y 488.291,Z 437.456,A -85,B 0,C 180,E1 -6355.479,E2 -6355.479} C_VEL
LIN {X 0,Y 488.2,Z 441.603,A -85,B 0,C 180,E1 -6356.268,E2 -6356.268} C_VEL
LIN {X 0,Y 488.046,Z 446.047,A -85,B 0,C 180,E1 -6357.317,E2 -6357.317} C_VEL
LIN {X 0,Y 488.024,Z 448.924,A -85,B 0,C 180,E1 -6358.174,E2 -6358.174} C_VEL
LIN {X 0,Y 487.967,Z 450.576,A -85,B 0,C 180,E1 -6358.77,E2 -6358.77} C_VEL
LIN {X 0,Y 487.881,Z 452.698,A -85,B 0,C 180,E1 -6359.804,E2 -6359.804} C_VEL
LIN {X 0,Y 487.823,Z 453.804,A -85,B 0,C 180,E1 -6360.671,E2 -6360.671} C_VEL
LIN {X 0,Y 487.83,Z 454.407,A -85,B 0,C 180,E1 -6361.614,E2 -6361.614} C_VEL
LIN {X 0,Y 487.787,Z 454.377,A -85,B 0,C 180,E1 -6362.546,E2 -6362.546} C_VEL
LIN {X 0,Y 487.814,Z 453.728,A -85,B 0,C 180,E1 -6363.474,E2 -6363.474} C_VEL
LIN {X 0,Y 487.848,Z 452.466,A -85,B 0,C 180,E1 -6364.395,E2 -6364.395} C_VEL
LIN {X 0,Y 487.958,Z 450.568,A -85,B 0,C 180,E1 -6365.312,E2 -6365.312} C_VEL
LIN {X 0,Y 488.057,Z 447.997,A -85,B 0,C 180,E1 -6366.222,E2 -6366.222} C_VEL
LIN {X 0,Y 488.106,Z 444.614,A -85,B 0,C 180,E1 -6367.147,E2 -6367.147} C_VEL
LIN {X 0,Y 488.251,Z 439.463,A -85,B 0,C 180,E1 -6368.245,E2 -6368.245} C_VEL
LIN {X 0,Y 488.426,Z 433.312,A -85,B 0,C 180,E1 -6369.275,E2 -6369.275} C_VEL
LIN {X 0,Y 488.596,Z 427.916,A -85,B 0,C 180,E1 -6370.025,E2 -6370.025} C_VEL
LIN {X 0,Y 488.852,Z 420.133,A -85,B 0,C 180,E1 -6370.91,E2 -6370.91} C_VEL
LIN {X 0,Y 489.06,Z 413.075,A -85,B 0,C 180,E1 -6371.57,E2 -6371.57} C_VEL
LIN {X 0,Y 489.298,Z 405.99,A -85,B 0,C 180,E1 -6372.121,E2 -6372.121} C_VEL
LIN {X 0,Y 489.516,Z 397.286,A -85,B 0,C 180,E1 -6372.669,E2 -6372.669} C_VEL
LIN {X 0,Y 489.703,Z 388.333,A -85,B 0,C 180,E1 -6373.106,E2 -6373.106} C_VEL
LIN {X 0,Y 489.86,Z 379.072,A -85,B 0,C 180,E1 -6373.439,E2 -6373.439} C_VEL
LIN {X 0,Y 489.999,Z 368.249,A -85,B 0,C 180,E1 -6373.692,E2 -6373.692} C_VEL
LIN {X 0,Y 490.261,Z 306.028,A -85,B 0,C 180,E1 -6374.613,E2 -6374.613} C_VEL
LIN {X 0,Y 488.607,Z 295.802,A -85,B 0,C 180,E1 -6374.819,E2 -6374.819} C_VEL
LIN {X 0,Y 488.858,Z 282.031,A -85,B 0,C 180,E1 -6378.012,E2 -6378.012} C_VEL
LIN {X 0,Y 489.007,Z 271.482,A -85,B 0,C 180,E1 -6380.487,E2 -6380.487} C_VEL
LIN {X 0,Y 488.858,Z 269.406,A -85,B 0,C 180,E1 -6381.006,E2 -6381.006} C_VEL
LIN {X 0,Y 488.82,Z 269.41,A -85,B 0,C 180,E1 -6383.395,E2 -6383.395} C_VEL
LIN {X 0,Y 488.697,Z 269.425,A -85,B 0,C 180,E1 -6385.877,E2 -6385.877} C_VEL
LIN {X 0,Y 488.962,Z 269.389,A -85,B 0,C 180,E1 -6387.529,E2 -6387.529} C_VEL
LIN {X 0,Y 488.936,Z 269.388,A -85,B 0,C 180,E1 -6390.824,E2 -6390.824} C_VEL
LIN {X 0,Y 488.963,Z 269.387,A -85,B 0,C 180,E1 -6392.471,E2 -6392.471} C_VEL
LIN {X 0,Y 488.84,Z 269.404,A -85,B 0,C 180,E1 -6395.776,E2 -6395.776} C_VEL
LIN {X 0,Y 488.818,Z 269.411,A -85,B 0,C 180,E1 -6398.266,E2 -6398.266} C_VEL
LIN {X 0,Y 488.807,Z 269.404,A -85,B 0,C 180,E1 -6401.612,E2 -6401.612} C_VEL
LIN {X 0,Y 488.763,Z 269.411,A -85,B 0,C 180,E1 -6405,E2 -6405} C_VEL
LIN {X 0,Y 488.747,Z 269.419,A -85,B 0,C 180,E1 -6408.442,E2 -6408.442} C_VEL
LIN {X 0,Y 488.707,Z 269.42,A -85,B 0,C 180,E1 -6411.07,E2 -6411.07} C_VEL
LIN {X 0,Y 488.687,Z 269.419,A -85,B 0,C 180,E1 -6413.745,E2 -6413.745} C_VEL
LIN {X 0,Y 488.79,Z 269.414,A -85,B 0,C 180,E1 -6416.943,E2 -6416.943} C_VEL
LIN {X 0,Y 488.707,Z 269.417,A -85,B 0,C 180,E1 -6420.362,E2 -6420.362} C_VEL
LIN {X 0,Y 488.726,Z 269.418,A -85,B 0,C 180,E1 -6423.482,E2 -6423.482} C_VEL
LIN {X 0,Y 488.678,Z 269.42,A -85,B 0,C 180,E1 -6426.353,E2 -6426.353} C_VEL
LIN {X 0,Y 488.696,Z 269.426,A -85,B 0,C 180,E1 -6429.253,E2 -6429.253} C_VEL
LIN {X 0,Y 488.701,Z 269.423,A -85,B 0,C 180,E1 -6431.599,E2 -6431.599} C_VEL
LIN {X 0,Y 488.706,Z 269.417,A -85,B 0,C 180,E1 -6434.8,E2 -6434.8} C_VEL
LIN {X 0,Y 488.725,Z 269.422,A -85,B 0,C 180,E1 -6437.478,E2 -6437.478} C_VEL
LIN {X 0,Y 488.735,Z 269.413,A -85,B 0,C 180,E1 -6440.749,E2 -6440.749} C_VEL
LIN {X 0,Y 488.677,Z 269.429,A -85,B 0,C 180,E1 -6443.868,E2 -6443.868} C_VEL
LIN {X 0,Y 488.73,Z 269.413,A -85,B 0,C 180,E1 -6446.876,E2 -6446.876} C_VEL
LIN {X 0,Y 488.724,Z 269.42,A -85,B 0,C 180,E1 -6449.781,E2 -6449.781} C_VEL
LIN {X 0,Y 488.789,Z 269.406,A -85,B 0,C 180,E1 -6453.054,E2 -6453.054} C_VEL
LIN {X 0,Y 488.682,Z 269.429,A -85,B 0,C 180,E1 -6456.254,E2 -6456.254} C_VEL
LIN {X 0,Y 488.734,Z 269.413,A -85,B 0,C 180,E1 -6459.175,E2 -6459.175} C_VEL
LIN {X 0,Y 488.722,Z 269.423,A -85,B 0,C 180,E1 -6462.423,E2 -6462.423} C_VEL
LIN {X 0,Y 488.749,Z 269.414,A -85,B 0,C 180,E1 -6464.999,E2 -6464.999} C_VEL
LIN {X 0,Y 488.792,Z 269.41,A -85,B 0,C 180,E1 -6468.387,E2 -6468.387} C_VEL
LIN {X 0,Y 488.804,Z 269.404,A -85,B 0,C 180,E1 -6471.733,E2 -6471.733} C_VEL
LIN {X 0,Y 488.835,Z 269.401,A -85,B 0,C 180,E1 -6474.224,E2 -6474.224} C_VEL
LIN {X 0,Y 488.946,Z 269.389,A -85,B 0,C 180,E1 -6477.528,E2 -6477.528} C_VEL
LIN {X 0,Y 488.963,Z 269.389,A -85,B 0,C 180,E1 -6480.823,E2 -6480.823} C_VEL
LIN {X 0,Y 488.947,Z 269.387,A -85,B 0,C 180,E1 -6482.471,E2 -6482.471} C_VEL
LIN {X 0,Y 488.841,Z 269.402,A -85,B 0,C 180,E1 -6485.776,E2 -6485.776} C_VEL
LIN {X 0,Y 488.804,Z 269.404,A -85,B 0,C 180,E1 -6488.267,E2 -6488.267} C_VEL
LIN {X 0,Y 488.819,Z 269.41,A -85,B 0,C 180,E1 -6491.612,E2 -6491.612} C_VEL
LIN {X 0,Y 488.748,Z 269.412,A -85,B 0,C 180,E1 -6495.001,E2 -6495.001} C_VEL
LIN {X 0,Y 488.742,Z 269.413,A -85,B 0,C 180,E1 -6498.443,E2 -6498.443} C_VEL
LIN {X 0,Y 488.694,Z 269.418,A -85,B 0,C 180,E1 -6501.071,E2 -6501.071} C_VEL
LIN {X 0,Y 488.681,Z 269.426,A -85,B 0,C 180,E1 -6503.746,E2 -6503.746} C_VEL
LIN {X 0,Y 488.78,Z 269.407,A -85,B 0,C 180,E1 -6506.944,E2 -6506.944} C_VEL
LIN {X 0,Y 488.698,Z 269.424,A -85,B 0,C 180,E1 -6510.363,E2 -6510.363} C_VEL
LIN {X 0,Y 488.725,Z 269.414,A -85,B 0,C 180,E1 -6513.485,E2 -6513.485} C_VEL
LIN {X 0,Y 488.677,Z 269.429,A -85,B 0,C 180,E1 -6516.356,E2 -6516.356} C_VEL
LIN {X 0,Y 488.69,Z 269.419,A -85,B 0,C 180,E1 -6519.255,E2 -6519.255} C_VEL
LIN {X 0,Y 488.699,Z 269.417,A -85,B 0,C 180,E1 -6521.601,E2 -6521.601} C_VEL
LIN {X 0,Y 488.693,Z 269.426,A -85,B 0,C 180,E1 -6524.804,E2 -6524.804} C_VEL
LIN {X 0,Y 488.681,Z 269.42,A -85,B 0,C 180,E1 -6527.475,E2 -6527.475} C_VEL
LIN {X 0,Y 488.694,Z 269.425,A -85,B 0,C 180,E1 -6530.747,E2 -6530.747} C_VEL
LIN {X 0,Y 488.671,Z 269.421,A -85,B 0,C 180,E1 -6533.869,E2 -6533.869} C_VEL
LIN {X 0,Y 488.73,Z 269.419,A -85,B 0,C 180,E1 -6536.878,E2 -6536.878} C_VEL
LIN {X 0,Y 488.717,Z 269.417,A -85,B 0,C 180,E1 -6539.781,E2 -6539.781} C_VEL
LIN {X 0,Y 488.698,Z 269.424,A -85,B 0,C 180,E1 -6543.078,E2 -6543.078} C_VEL
LIN {X 0,Y 488.679,Z 269.423,A -85,B 0,C 180,E1 -6546.255,E2 -6546.255} C_VEL
LIN {X 0,Y 488.762,Z 269.559,A -85,B 0,C 180,E1 -6546.906,E2 -6546.906} C_VEL
LIN {X 0,Y 489.84,Z 276.359,A -85,B 0,C 180,E1 -6548.341,E2 -6548.341} C_VEL
LIN {X 0,Y 489.375,Z 290.311,A -85,B 0,C 180,E1 -6551.133,E2 -6551.133} C_VEL
LIN {X 0,Y 488.944,Z 306.74,A -85,B 0,C 180,E1 -6554.375,E2 -6554.375} C_VEL
LIN {X 0,Y 488.552,Z 321.382,A -85,B 0,C 180,E1 -6557.22,E2 -6557.22} C_VEL
LIN {X 0,Y 490.267,Z 335.036,A -85,B 0,C 180,E1 -6557.467,E2 -6557.467} C_VEL
LIN {X 0,Y 489.937,Z 398.064,A -85,B 0,C 180,E1 -6558.415,E2 -6558.415} C_VEL
LIN {X 0,Y 489.696,Z 407.951,A -85,B 0,C 180,E1 -6558.671,E2 -6558.671} C_VEL
LIN {X 0,Y 489.508,Z 418.527,A -85,B 0,C 180,E1 -6559.086,E2 -6559.086} C_VEL
LIN {X 0,Y 489.243,Z 428.89,A -85,B 0,C 180,E1 -6559.656,E2 -6559.656} C_VEL
LIN {X 0,Y 488.978,Z 438.765,A -85,B 0,C 180,E1 -6560.382,E2 -6560.382} C_VEL
LIN {X 0,Y 488.711,Z 446.678,A -85,B 0,C 180,E1 -6561.107,E2 -6561.107} C_VEL
LIN {X 0,Y 488.431,Z 454.073,A -85,B 0,C 180,E1 -6561.935,E2 -6561.935} C_VEL
LIN {X 0,Y 488.276,Z 461.581,A -85,B 0,C 180,E1 -6562.973,E2 -6562.973} C_VEL
LIN {X 0,Y 488.136,Z 468.434,A -85,B 0,C 180,E1 -6564.216,E2 -6564.216} C_VEL
LIN {X 0,Y 487.953,Z 473.628,A -85,B 0,C 180,E1 -6565.457,E2 -6565.457} C_VEL
LIN {X 0,Y 487.985,Z 477.446,A -85,B 0,C 180,E1 -6566.698,E2 -6566.698} C_VEL
LIN {X 0,Y 487.911,Z 479.201,A -85,B 0,C 180,E1 -6567.523,E2 -6567.523} C_VEL
LIN {X 0,Y 487.889,Z 480.458,A -85,B 0,C 180,E1 -6568.349,E2 -6568.349} C_VEL
LIN {X 0,Y 487.831,Z 481.239,A -85,B 0,C 180,E1 -6569.175,E2 -6569.175} C_VEL
LIN {X 0,Y 487.818,Z 481.532,A -85,B 0,C 180,E1 -6570,E2 -6570} C_VEL
LIN {X 0,Y 487.831,Z 481.233,A -85,B 0,C 180,E1 -6570.825,E2 -6570.825} C_VEL
LIN {X 0,Y 487.889,Z 480.447,A -85,B 0,C 180,E1 -6571.651,E2 -6571.651} C_VEL
LIN {X 0,Y 487.911,Z 479.185,A -85,B 0,C 180,E1 -6572.477,E2 -6572.477} C_VEL
LIN {X 0,Y 488.007,Z 476.267,A -85,B 0,C 180,E1 -6573.716,E2 -6573.716} C_VEL
LIN {X 0,Y 487.953,Z 473.603,A -85,B 0,C 180,E1 -6574.543,E2 -6574.543} C_VEL
LIN {X 0,Y 488.134,Z 468.4,A -85,B 0,C 180,E1 -6575.784,E2 -6575.784} C_VEL
LIN {X 0,Y 488.277,Z 461.537,A -85,B 0,C 180,E1 -6577.027,E2 -6577.027} C_VEL
LIN {X 0,Y 488.43,Z 454.039,A -85,B 0,C 180,E1 -6578.064,E2 -6578.064} C_VEL
LIN {X 0,Y 488.711,Z 446.648,A -85,B 0,C 180,E1 -6578.893,E2 -6578.893} C_VEL
LIN {X 0,Y 488.977,Z 438.732,A -85,B 0,C 180,E1 -6579.618,E2 -6579.618} C_VEL
LIN {X 0,Y 489.194,Z 430.364,A -85,B 0,C 180,E1 -6580.24,E2 -6580.24} C_VEL
LIN {X 0,Y 489.48,Z 419.664,A -85,B 0,C 180,E1 -6580.862,E2 -6580.862} C_VEL
LIN {X 0,Y 489.646,Z 408.811,A -85,B 0,C 180,E1 -6581.303,E2 -6581.303} C_VEL
LIN {X 0,Y 489.893,Z 399.45,A -85,B 0,C 180,E1 -6581.56,E2 -6581.56} C_VEL
LIN {X 0,Y 490.129,Z 372.212,A -85,B 0,C 180,E1 -6581.986,E2 -6581.986} C_VEL
LIN {X 0,Y 490.088,Z 332.967,A -85,B 0,C 180,E1 -6582.57,E2 -6582.57} C_VEL
LIN {X 0,Y 488.546,Z 321.095,A -85,B 0,C 180,E1 -6582.789,E2 -6582.789} C_VEL
LIN {X 0,Y 488.918,Z 305.172,A -85,B 0,C 180,E1 -6585.849,E2 -6585.849} C_VEL
LIN {X 0,Y 489.257,Z 289.928,A -85,B 0,C 180,E1 -6588.813,E2 -6588.813} C_VEL
LIN {X 0,Y 489.682,Z 276.409,A -85,B 0,C 180,E1 -6591.467,E2 -6591.467} C_VEL
LIN {X 0,Y 488.761,Z 269.418,A -85,B 0,C 180,E1 -6592.912,E2 -6592.912} C_VEL
LIN {X 0,Y 488.689,Z 269.422,A -85,B 0,C 180,E1 -6595.558,E2 -6595.558} C_VEL
LIN {X 0,Y 488.681,Z 269.429,A -85,B 0,C 180,E1 -6598.685,E2 -6598.685} C_VEL
LIN {X 0,Y 488.684,Z 269.424,A -85,B 0,C 180,E1 -6601.179,E2 -6601.179} C_VEL
LIN {X 0,Y 488.718,Z 269.416,A -85,B 0,C 180,E1 -6604.113,E2 -6604.113} C_VEL
LIN {X 0,Y 488.673,Z 269.431,A -85,B 0,C 180,E1 -6607.158,E2 -6607.158} C_VEL
LIN {X 0,Y 488.712,Z 269.419,A -85,B 0,C 180,E1 -6610.344,E2 -6610.344} C_VEL
LIN {X 0,Y 488.67,Z 269.427,A -85,B 0,C 180,E1 -6613.655,E2 -6613.655} C_VEL
LIN {X 0,Y 488.676,Z 269.422,A -85,B 0,C 180,E1 -6616.344,E2 -6616.344} C_VEL
LIN {X 0,Y 488.724,Z 269.422,A -85,B 0,C 180,E1 -6619.676,E2 -6619.676} C_VEL
LIN {X 0,Y 488.671,Z 269.419,A -85,B 0,C 180,E1 -6622.84,E2 -6622.84} C_VEL
LIN {X 0,Y 488.721,Z 269.42,A -85,B 0,C 180,E1 -6625.887,E2 -6625.887} C_VEL
LIN {X 0,Y 488.68,Z 269.419,A -85,B 0,C 180,E1 -6628.82,E2 -6628.82} C_VEL
LIN {X 0,Y 488.731,Z 269.419,A -85,B 0,C 180,E1 -6631.671,E2 -6631.671} C_VEL
LIN {X 0,Y 488.74,Z 269.411,A -85,B 0,C 180,E1 -6633.527,E2 -6633.527} C_VEL
LIN {X 0,Y 488.667,Z 269.426,A -85,B 0,C 180,E1 -6636.253,E2 -6636.253} C_VEL
LIN {X 0,Y 488.733,Z 269.41,A -85,B 0,C 180,E1 -6639.175,E2 -6639.175} C_VEL
LIN {X 0,Y 488.747,Z 269.413,A -85,B 0,C 180,E1 -6641.627,E2 -6641.627} C_VEL
LIN {X 0,Y 488.747,Z 269.41,A -85,B 0,C 180,E1 -6644.999,E2 -6644.999} C_VEL
LIN {X 0,Y 488.795,Z 269.413,A -85,B 0,C 180,E1 -6648.387,E2 -6648.387} C_VEL
LIN {X 0,Y 488.803,Z 269.401,A -85,B 0,C 180,E1 -6651.733,E2 -6651.733} C_VEL
LIN {X 0,Y 488.84,Z 269.402,A -85,B 0,C 180,E1 -6654.224,E2 -6654.224} C_VEL
LIN {X 0,Y 488.946,Z 269.385,A -85,B 0,C 180,E1 -6657.529,E2 -6657.529} C_VEL
LIN {X 0,Y 488.952,Z 269.385,A -85,B 0,C 180,E1 -6660,E2 -6660} C_VEL
LIN {X 0,Y 488.945,Z 269.384,A -85,B 0,C 180,E1 -6662.472,E2 -6662.472} C_VEL
LIN {X 0,Y 488.828,Z 269.402,A -85,B 0,C 180,E1 -6665.776,E2 -6665.776} C_VEL
LIN {X 0,Y 488.804,Z 269.402,A -85,B 0,C 180,E1 -6668.267,E2 -6668.267} C_VEL
LIN {X 0,Y 488.792,Z 269.408,A -85,B 0,C 180,E1 -6671.613,E2 -6671.613} C_VEL
LIN {X 0,Y 488.749,Z 269.415,A -85,B 0,C 180,E1 -6675.001,E2 -6675.001} C_VEL
LIN {X 0,Y 488.743,Z 269.414,A -85,B 0,C 180,E1 -6678.443,E2 -6678.443} C_VEL
LIN {X 0,Y 488.695,Z 269.419,A -85,B 0,C 180,E1 -6681.071,E2 -6681.071} C_VEL
LIN {X 0,Y 488.682,Z 269.428,A -85,B 0,C 180,E1 -6683.746,E2 -6683.746} C_VEL
LIN {X 0,Y 488.788,Z 269.406,A -85,B 0,C 180,E1 -6686.946,E2 -6686.946} C_VEL
LIN {X 0,Y 488.708,Z 269.421,A -85,B 0,C 180,E1 -6690.365,E2 -6690.365} C_VEL
LIN {X 0,Y 488.726,Z 269.417,A -85,B 0,C 180,E1 -6693.485,E2 -6693.485} C_VEL
LIN {X 0,Y 488.681,Z 269.428,A -85,B 0,C 180,E1 -6696.357,E2 -6696.357} C_VEL
LIN {X 0,Y 488.734,Z 269.415,A -85,B 0,C 180,E1 -6699.251,E2 -6699.251} C_VEL
LIN {X 0,Y 488.737,Z 269.422,A -85,B 0,C 180,E1 -6702.521,E2 -6702.521} C_VEL
LIN {X 0,Y 488.813,Z 269.591,A -85,B 0,C 180,E1 -6703.742,E2 -6703.742} C_VEL
LIN {X 0,Y 488.736,Z 282.941,A -85,B 0,C 180,E1 -6706.578,E2 -6706.578} C_VEL
LIN {X 0,Y 488.657,Z 295.48,A -85,B 0,C 180,E1 -6709.262,E2 -6709.262} C_VEL
LIN {X 0,Y 490.348,Z 307.563,A -85,B 0,C 180,E1 -6709.496,E2 -6709.496} C_VEL
LIN {X 0,Y 489.944,Z 372.073,A -85,B 0,C 180,E1 -6710.468,E2 -6710.468} C_VEL
LIN {X 0,Y 489.82,Z 382.512,A -85,B 0,C 180,E1 -6710.751,E2 -6710.751} C_VEL
LIN {X 0,Y 489.609,Z 394.006,A -85,B 0,C 180,E1 -6711.231,E2 -6711.231} C_VEL
LIN {X 0,Y 489.344,Z 402.926,A -85,B 0,C 180,E1 -6711.746,E2 -6711.746} C_VEL
LIN {X 0,Y 488.588,Z 408.218,A -85,B 0,C 180,E1 -6712.099,E2 -6712.099} C_VEL
LIN {X 0,Y 485.471,Z 416.206,A -85,B 0,C 180,E1 -6712.699,E2 -6712.699} C_VEL
LIN {X 0,Y 482.382,Z 423.453,A -85,B 0,C 180,E1 -6713.378,E2 -6713.378} C_VEL
LIN {X 0,Y 481.597,Z 427.528,A -85,B 0,C 180,E1 -6713.864,E2 -6713.864} C_VEL
LIN {X 0,Y 481.368,Z 434.506,A -85,B 0,C 180,E1 -6714.846,E2 -6714.846} C_VEL
LIN {X 0,Y 481.183,Z 441.141,A -85,B 0,C 180,E1 -6716.038,E2 -6716.038} C_VEL
LIN {X 0,Y 481.017,Z 444.677,A -85,B 0,C 180,E1 -6716.82,E2 -6716.82} C_VEL
LIN {X 0,Y 480.953,Z 448.652,A -85,B 0,C 180,E1 -6717.945,E2 -6717.945} C_VEL
LIN {X 0,Y 480.821,Z 451.861,A -85,B 0,C 180,E1 -6719.232,E2 -6719.232} C_VEL
LIN {X 0,Y 480.749,Z 453.484,A -85,B 0,C 180,E1 -6720.197,E2 -6720.197} C_VEL
LIN {X 0,Y 480.721,Z 454.49,A -85,B 0,C 180,E1 -6721.305,E2 -6721.305} C_VEL
LIN {X 0,Y 480.7,Z 454.737,A -85,B 0,C 180,E1 -6722.106,E2 -6722.106} C_VEL
LIN {X 0,Y 480.699,Z 454.338,A -85,B 0,C 180,E1 -6723.106,E2 -6723.106} C_VEL
LIN {X 0,Y 480.726,Z 453.355,A -85,B 0,C 180,E1 -6723.987,E2 -6723.987} C_VEL
LIN {X 0,Y 480.892,Z 450.588,A -85,B 0,C 180,E1 -6725.422,E2 -6725.422} C_VEL
LIN {X 0,Y 480.992,Z 448.101,A -85,B 0,C 180,E1 -6726.309,E2 -6726.309} C_VEL
LIN {X 0,Y 481.103,Z 442.769,A -85,B 0,C 180,E1 -6727.679,E2 -6727.679} C_VEL
LIN {X 0,Y 481.21,Z 438.254,A -85,B 0,C 180,E1 -6728.586,E2 -6728.586} C_VEL
LIN {X 0,Y 481.403,Z 432.753,A -85,B 0,C 180,E1 -6729.49,E2 -6729.49} C_VEL
LIN {X 0,Y 481.558,Z 427.9,A -85,B 0,C 180,E1 -6730.165,E2 -6730.165} C_VEL
LIN {X 0,Y 481.829,Z 421.143,A -85,B 0,C 180,E1 -6730.952,E2 -6730.952} C_VEL
LIN {X 0,Y 482.053,Z 414.053,A -85,B 0,C 180,E1 -6731.639,E2 -6731.639} C_VEL
LIN {X 0,Y 482.32,Z 405.801,A -85,B 0,C 180,E1 -6732.292,E2 -6732.292} C_VEL
LIN {X 0,Y 482.567,Z 396.985,A -85,B 0,C 180,E1 -6732.848,E2 -6732.848} C_VEL
LIN {X 0,Y 482.76,Z 388.006,A -85,B 0,C 180,E1 -6733.286,E2 -6733.286} C_VEL
LIN {X 0,Y 482.961,Z 377.201,A -85,B 0,C 180,E1 -6733.667,E2 -6733.667} C_VEL
LIN {X 0,Y 483.103,Z 362.214,A -85,B 0,C 180,E1 -6733.955,E2 -6733.955} C_VEL
LIN {X 0,Y 483.331,Z 306.81,A -85,B 0,C 180,E1 -6734.784,E2 -6734.784} C_VEL
LIN {X 0,Y 481.604,Z 295.908,A -85,B 0,C 180,E1 -6735.015,E2 -6735.015} C_VEL
LIN {X 0,Y 481.887,Z 282.266,A -85,B 0,C 180,E1 -6738.219,E2 -6738.219} C_VEL
LIN {X 0,Y 482.021,Z 273.295,A -85,B 0,C 180,E1 -6740.348,E2 -6740.348} C_VEL
LIN {X 0,Y 481.842,Z 270.28,A -85,B 0,C 180,E1 -6741.085,E2 -6741.085} C_VEL
LIN {X 0,Y 481.809,Z 270.28,A -85,B 0,C 180,E1 -6744.14,E2 -6744.14} C_VEL
LIN {X 0,Y 481.929,Z 270.265,A -85,B 0,C 180,E1 -6747.493,E2 -6747.493} C_VEL
LIN {X 0,Y 481.888,Z 270.266,A -85,B 0,C 180,E1 -6750.836,E2 -6750.836} C_VEL
LIN {X 0,Y 481.93,Z 270.263,A -85,B 0,C 180,E1 -6752.507,E2 -6752.507} C_VEL
LIN {X 0,Y 481.799,Z 270.282,A -85,B 0,C 180,E1 -6755.86,E2 -6755.86} C_VEL
LIN {X 0,Y 481.763,Z 270.288,A -85,B 0,C 180,E1 -6758.388,E2 -6758.388} C_VEL
LIN {X 0,Y 481.752,Z 270.285,A -85,B 0,C 180,E1 -6761.785,E2 -6761.785} C_VEL
LIN {X 0,Y 481.744,Z 270.284,A -85,B 0,C 180,E1 -6765.224,E2 -6765.224} C_VEL
LIN {X 0,Y 481.709,Z 270.295,A -85,B 0,C 180,E1 -6768.721,E2 -6768.721} C_VEL
LIN {X 0,Y 481.645,Z 270.297,A -85,B 0,C 180,E1 -6771.394,E2 -6771.394} C_VEL
LIN {X 0,Y 481.672,Z 270.294,A -85,B 0,C 180,E1 -6774.113,E2 -6774.113} C_VEL
LIN {X 0,Y 481.745,Z 270.289,A -85,B 0,C 180,E1 -6777.138,E2 -6777.138} C_VEL
LIN {X 0,Y 481.677,Z 270.292,A -85,B 0,C 180,E1 -6779.74,E2 -6779.74} C_VEL
LIN {X 0,Y 481.667,Z 270.297,A -85,B 0,C 180,E1 -6782.673,E2 -6782.673} C_VEL
LIN {X 0,Y 481.632,Z 270.3,A -85,B 0,C 180,E1 -6785.709,E2 -6785.709} C_VEL
LIN {X 0,Y 481.666,Z 270.296,A -85,B 0,C 180,E1 -6788.858,E2 -6788.858} C_VEL
LIN {X 0,Y 481.647,Z 270.298,A -85,B 0,C 180,E1 -6791.912,E2 -6791.912} C_VEL
LIN {X 0,Y 481.654,Z 270.295,A -85,B 0,C 180,E1 -6794.456,E2 -6794.456} C_VEL
LIN {X 0,Y 481.682,Z 270.292,A -85,B 0,C 180,E1 -6796.845,E2 -6796.845} C_VEL
LIN {X 0,Y 481.682,Z 270.295,A -85,B 0,C 180,E1 -6800.06,E2 -6800.06} C_VEL
LIN {X 0,Y 481.621,Z 270.301,A -85,B 0,C 180,E1 -6803.252,E2 -6803.252} C_VEL
LIN {X 0,Y 481.701,Z 270.292,A -85,B 0,C 180,E1 -6806.329,E2 -6806.329} C_VEL
LIN {X 0,Y 481.648,Z 270.297,A -85,B 0,C 180,E1 -6809.415,E2 -6809.415} C_VEL
LIN {X 0,Y 481.693,Z 270.299,A -85,B 0,C 180,E1 -6812.167,E2 -6812.167} C_VEL
LIN {X 0,Y 481.707,Z 270.289,A -85,B 0,C 180,E1 -6814.969,E2 -6814.969} C_VEL
LIN {X 0,Y 481.638,Z 270.298,A -85,B 0,C 180,E1 -6817.704,E2 -6817.704} C_VEL
LIN {X 0,Y 481.694,Z 270.299,A -85,B 0,C 180,E1 -6820.392,E2 -6820.392} C_VEL
LIN {X 0,Y 481.679,Z 270.294,A -85,B 0,C 180,E1 -6823.033,E2 -6823.033} C_VEL
LIN {X 0,Y 481.676,Z 270.292,A -85,B 0,C 180,E1 -6825.638,E2 -6825.638} C_VEL
LIN {X 0,Y 481.738,Z 270.287,A -85,B 0,C 180,E1 -6828.215,E2 -6828.215} C_VEL
LIN {X 0,Y 481.75,Z 270.283,A -85,B 0,C 180,E1 -6831.611,E2 -6831.611} C_VEL
LIN {X 0,Y 481.795,Z 270.278,A -85,B 0,C 180,E1 -6834.139,E2 -6834.139} C_VEL
LIN {X 0,Y 481.913,Z 270.265,A -85,B 0,C 180,E1 -6837.492,E2 -6837.492} C_VEL
LIN {X 0,Y 481.913,Z 270.267,A -85,B 0,C 180,E1 -6840.836,E2 -6840.836} C_VEL
LIN {X 0,Y 481.914,Z 270.263,A -85,B 0,C 180,E1 -6842.507,E2 -6842.507} C_VEL
LIN {X 0,Y 481.8,Z 270.279,A -85,B 0,C 180,E1 -6845.861,E2 -6845.861} C_VEL
LIN {X 0,Y 481.749,Z 270.283,A -85,B 0,C 180,E1 -6848.388,E2 -6848.388} C_VEL
LIN {X 0,Y 481.783,Z 270.284,A -85,B 0,C 180,E1 -6851.784,E2 -6851.784} C_VEL
LIN {X 0,Y 481.729,Z 270.289,A -85,B 0,C 180,E1 -6855.225,E2 -6855.225} C_VEL
LIN {X 0,Y 481.699,Z 270.289,A -85,B 0,C 180,E1 -6858.722,E2 -6858.722} C_VEL
LIN {X 0,Y 481.633,Z 270.3,A -85,B 0,C 180,E1 -6861.395,E2 -6861.395} C_VEL
LIN {X 0,Y 481.665,Z 270.3,A -85,B 0,C 180,E1 -6864.114,E2 -6864.114} C_VEL
LIN {X 0,Y 481.734,Z 270.285,A -85,B 0,C 180,E1 -6867.14,E2 -6867.14} C_VEL
LIN {X 0,Y 481.667,Z 270.296,A -85,B 0,C 180,E1 -6869.742,E2 -6869.742} C_VEL
LIN {X 0,Y 481.661,Z 270.297,A -85,B 0,C 180,E1 -6872.675,E2 -6872.675} C_VEL
LIN {X 0,Y 481.631,Z 270.299,A -85,B 0,C 180,E1 -6875.71,E2 -6875.71} C_VEL
LIN {X 0,Y 481.66,Z 270.298,A -85,B 0,C 180,E1 -6878.86,E2 -6878.86} C_VEL
LIN {X 0,Y 481.644,Z 270.297,A -85,B 0,C 180,E1 -6881.914,E2 -6881.914} C_VEL
LIN {X 0,Y 481.647,Z 270.302,A -85,B 0,C 180,E1 -6884.459,E2 -6884.459} C_VEL
LIN {X 0,Y 481.635,Z 270.297,A -85,B 0,C 180,E1 -6887.84,E2 -6887.84} C_VEL
LIN {X 0,Y 481.653,Z 270.3,A -85,B 0,C 180,E1 -6890.655,E2 -6890.655} C_VEL
LIN {X 0,Y 481.621,Z 270.303,A -85,B 0,C 180,E1 -6893.377,E2 -6893.377} C_VEL
LIN {X 0,Y 481.671,Z 270.293,A -85,B 0,C 180,E1 -6896.328,E2 -6896.328} C_VEL
LIN {X 0,Y 481.644,Z 270.302,A -85,B 0,C 180,E1 -6899.419,E2 -6899.419} C_VEL
LIN {X 0,Y 481.657,Z 270.296,A -85,B 0,C 180,E1 -6902.166,E2 -6902.166} C_VEL
LIN {X 0,Y 481.67,Z 270.298,A -85,B 0,C 180,E1 -6904.968,E2 -6904.968} C_VEL
LIN {X 0,Y 481.712,Z 270.298,A -85,B 0,C 180,E1 -6906.742,E2 -6906.742} C_VEL
LIN {X 0,Y 482.858,Z 278.243,A -85,B 0,C 180,E1 -6908.438,E2 -6908.438} C_VEL
LIN {X 0,Y 482.269,Z 294.553,A -85,B 0,C 180,E1 -6911.741,E2 -6911.741} C_VEL
LIN {X 0,Y 481.809,Z 309.754,A -85,B 0,C 180,E1 -6914.778,E2 -6914.778} C_VEL
LIN {X 0,Y 481.517,Z 321.136,A -85,B 0,C 180,E1 -6917.03,E2 -6917.03} C_VEL
LIN {X 0,Y 483.318,Z 335.286,A -85,B 0,C 180,E1 -6917.293,E2 -6917.293} C_VEL
LIN {X 0,Y 483,Z 397.723,A -85,B 0,C 180,E1 -6918.246,E2 -6918.246} C_VEL
LIN {X 0,Y 482.753,Z 406.829,A -85,B 0,C 180,E1 -6918.48,E2 -6918.48} C_VEL
LIN {X 0,Y 482.587,Z 415.842,A -85,B 0,C 180,E1 -6918.821,E2 -6918.821} C_VEL
LIN {X 0,Y 482.314,Z 425.118,A -85,B 0,C 180,E1 -6919.293,E2 -6919.293} C_VEL
LIN {X 0,Y 482.014,Z 436.057,A -85,B 0,C 180,E1 -6920.03,E2 -6920.03} C_VEL
LIN {X 0,Y 481.703,Z 445.43,A -85,B 0,C 180,E1 -6920.871,E2 -6920.871} C_VEL
LIN {X 0,Y 481.457,Z 452.145,A -85,B 0,C 180,E1 -6921.607,E2 -6921.607} C_VEL
LIN {X 0,Y 481.235,Z 458.516,A -85,B 0,C 180,E1 -6922.448,E2 -6922.448} C_VEL
LIN {X 0,Y 481.152,Z 464.083,A -85,B 0,C 180,E1 -6923.338,E2 -6923.338} C_VEL
LIN {X 0,Y 481.047,Z 468.227,A -85,B 0,C 180,E1 -6924.13,E2 -6924.13} C_VEL
LIN {X 0,Y 480.87,Z 473.425,A -85,B 0,C 180,E1 -6925.39,E2 -6925.39} C_VEL
LIN {X 0,Y 480.914,Z 477.245,A -85,B 0,C 180,E1 -6926.649,E2 -6926.649} C_VEL
LIN {X 0,Y 480.826,Z 479.002,A -85,B 0,C 180,E1 -6927.487,E2 -6927.487} C_VEL
LIN {X 0,Y 480.791,Z 480.261,A -85,B 0,C 180,E1 -6928.325,E2 -6928.325} C_VEL
LIN {X 0,Y 480.757,Z 481.043,A -85,B 0,C 180,E1 -6929.162,E2 -6929.162} C_VEL
LIN {X 0,Y 480.742,Z 481.337,A -85,B 0,C 180,E1 -6930,E2 -6930} C_VEL
LIN {X 0,Y 480.757,Z 481.037,A -85,B 0,C 180,E1 -6930.838,E2 -6930.838} C_VEL
LIN {X 0,Y 480.791,Z 480.252,A -85,B 0,C 180,E1 -6931.675,E2 -6931.675} C_VEL
LIN {X 0,Y 480.826,Z 478.99,A -85,B 0,C 180,E1 -6932.513,E2 -6932.513} C_VEL
LIN {X 0,Y 480.91,Z 476.07,A -85,B 0,C 180,E1 -6933.771,E2 -6933.771} C_VEL
LIN {X 0,Y 480.87,Z 473.406,A -85,B 0,C 180,E1 -6934.61,E2 -6934.61} C_VEL
LIN {X 0,Y 481.038,Z 468.2,A -85,B 0,C 180,E1 -6935.87,E2 -6935.87} C_VEL
LIN {X 0,Y 481.205,Z 461.337,A -85,B 0,C 180,E1 -6937.131,E2 -6937.131} C_VEL
LIN {X 0,Y 481.39,Z 453.838,A -85,B 0,C 180,E1 -6938.183,E2 -6938.183} C_VEL
LIN {X 0,Y 481.692,Z 446.445,A -85,B 0,C 180,E1 -6939.024,E2 -6939.024} C_VEL
LIN {X 0,Y 481.971,Z 438.527,A -85,B 0,C 180,E1 -6939.759,E2 -6939.759} C_VEL
LIN {X 0,Y 482.194,Z 430.158,A -85,B 0,C 180,E1 -6940.391,E2 -6940.391} C_VEL
LIN {X 0,Y 482.509,Z 419.456,A -85,B 0,C 180,E1 -6941.021,E2 -6941.021} C_VEL
LIN {X 0,Y 482.691,Z 408.601,A -85,B 0,C 180,E1 -6941.468,E2 -6941.468} C_VEL
LIN {X 0,Y 482.949,Z 399.238,A -85,B 0,C 180,E1 -6941.728,E2 -6941.728} C_VEL
LIN {X 0,Y 483.221,Z 367.88,A -85,B 0,C 180,E1 -6942.223,E2 -6942.223} C_VEL
LIN {X 0,Y 483.192,Z 333.884,A -85,B 0,C 180,E1 -6942.736,E2 -6942.736} C_VEL
LIN {X 0,Y 481.517,Z 320.795,A -85,B 0,C 180,E1 -6942.997,E2 -6942.997} C_VEL
LIN {X 0,Y 481.911,Z 304.98,A -85,B 0,C 180,E1 -6946.086,E2 -6946.086} C_VEL
LIN {X 0,Y 482.237,Z 290.598,A -85,B 0,C 180,E1 -6948.92,E2 -6948.92} C_VEL
LIN {X 0,Y 482.683,Z 277.285,A -85,B 0,C 180,E1 -6951.57,E2 -6951.57} C_VEL
LIN {X 0,Y 481.705,Z 270.297,A -85,B 0,C 180,E1 -6953.03,E2 -6953.03} C_VEL
LIN {X 0,Y 481.641,Z 270.301,A -85,B 0,C 180,E1 -6955.96,E2 -6955.96} C_VEL
LIN {X 0,Y 481.636,Z 270.305,A -85,B 0,C 180,E1 -6958.894,E2 -6958.894} C_VEL
LIN {X 0,Y 481.651,Z 270.297,A -85,B 0,C 180,E1 -6962.188,E2 -6962.188} C_VEL
LIN {X 0,Y 481.654,Z 270.303,A -85,B 0,C 180,E1 -6965.203,E2 -6965.203} C_VEL
LIN {X 0,Y 481.648,Z 270.299,A -85,B 0,C 180,E1 -6968.006,E2 -6968.006} C_VEL
LIN {X 0,Y 481.64,Z 270.308,A -85,B 0,C 180,E1 -6971.042,E2 -6971.042} C_VEL
LIN {X 0,Y 481.646,Z 270.299,A -85,B 0,C 180,E1 -6974.457,E2 -6974.457} C_VEL
LIN {X 0,Y 481.639,Z 270.3,A -85,B 0,C 180,E1 -6977.838,E2 -6977.838} C_VEL
LIN {X 0,Y 481.65,Z 270.296,A -85,B 0,C 180,E1 -6980.653,E2 -6980.653} C_VEL
LIN {X 0,Y 481.62,Z 270.302,A -85,B 0,C 180,E1 -6983.375,E2 -6983.375} C_VEL
LIN {X 0,Y 481.7,Z 270.289,A -85,B 0,C 180,E1 -6986.329,E2 -6986.329} C_VEL
LIN {X 0,Y 481.639,Z 270.3,A -85,B 0,C 180,E1 -6989.417,E2 -6989.417} C_VEL
LIN {X 0,Y 481.687,Z 270.292,A -85,B 0,C 180,E1 -6992.167,E2 -6992.167} C_VEL
LIN {X 0,Y 481.68,Z 270.292,A -85,B 0,C 180,E1 -6994.968,E2 -6994.968} C_VEL
LIN {X 0,Y 481.635,Z 270.299,A -85,B 0,C 180,E1 -6997.704,E2 -6997.704} C_VEL
LIN {X 0,Y 481.692,Z 270.298,A -85,B 0,C 180,E1 -7000.393,E2 -7000.393} C_VEL
LIN {X 0,Y 481.673,Z 270.291,A -85,B 0,C 180,E1 -7003.033,E2 -7003.033} C_VEL
LIN {X 0,Y 481.673,Z 270.29,A -85,B 0,C 180,E1 -7005.638,E2 -7005.638} C_VEL
LIN {X 0,Y 481.739,Z 270.289,A -85,B 0,C 180,E1 -7008.215,E2 -7008.215} C_VEL
LIN {X 0,Y 481.749,Z 270.28,A -85,B 0,C 180,E1 -7011.612,E2 -7011.612} C_VEL
LIN {X 0,Y 481.799,Z 270.278,A -85,B 0,C 180,E1 -7014.139,E2 -7014.139} C_VEL
LIN {X 0,Y 481.913,Z 270.261,A -85,B 0,C 180,E1 -7017.493,E2 -7017.493} C_VEL
LIN {X 0,Y 481.892,Z 270.272,A -85,B 0,C 180,E1 -7020.836,E2 -7020.836} C_VEL
LIN {X 0,Y 481.913,Z 270.26,A -85,B 0,C 180,E1 -7022.508,E2 -7022.508} C_VEL
LIN {X 0,Y 481.786,Z 270.279,A -85,B 0,C 180,E1 -7025.861,E2 -7025.861} C_VEL
LIN {X 0,Y 481.749,Z 270.281,A -85,B 0,C 180,E1 -7028.389,E2 -7028.389} C_VEL
LIN {X 0,Y 481.737,Z 270.285,A -85,B 0,C 180,E1 -7031.785,E2 -7031.785} C_VEL
LIN {X 0,Y 481.729,Z 270.292,A -85,B 0,C 180,E1 -7035.225,E2 -7035.225} C_VEL
LIN {X 0,Y 481.7,Z 270.291,A -85,B 0,C 180,E1 -7038.722,E2 -7038.722} C_VEL
LIN {X 0,Y 481.634,Z 270.302,A -85,B 0,C 180,E1 -7041.395,E2 -7041.395} C_VEL
LIN {X 0,Y 481.666,Z 270.3,A -85,B 0,C 180,E1 -7044.114,E2 -7044.114} C_VEL
LIN {X 0,Y 481.742,Z 270.285,A -85,B 0,C 180,E1 -7047.141,E2 -7047.141} C_VEL
LIN {X 0,Y 481.677,Z 270.297,A -85,B 0,C 180,E1 -7049.741,E2 -7049.741} C_VEL
LIN {X 0,Y 481.663,Z 270.297,A -85,B 0,C 180,E1 -7052.675,E2 -7052.675} C_VEL
LIN {X 0,Y 481.635,Z 270.299,A -85,B 0,C 180,E1 -7055.71,E2 -7055.71} C_VEL
LIN {X 0,Y 481.706,Z 270.291,A -85,B 0,C 180,E1 -7059.355,E2 -7059.355} C_VEL
LIN {X 0,Y 481.673,Z 270.3,A -85,B 0,C 180,E1 -7062.158,E2 -7062.158} C_VEL
LIN {X 0,Y 481.79,Z 270.452,A -85,B 0,C 180,E1 -7063.643,E2 -7063.643} C_VEL
LIN {X 0,Y 481.725,Z 283.45,A -85,B 0,C 180,E1 -7066.442,E2 -7066.442} C_VEL
LIN {X 0,Y 481.604,Z 295.597,A -85,B 0,C 180,E1 -7069.059,E2 -7069.059} C_VEL
LIN {X 0,Y 483.431,Z 307.645,A -85,B 0,C 180,E1 -7069.311,E2 -7069.311} C_VEL
LIN {X 0,Y 483.016,Z 371.656,A -85,B 0,C 180,E1 -7070.287,E2 -7070.287} C_VEL
LIN {X 0,Y 482.887,Z 380.837,A -85,B 0,C 180,E1 -7070.527,E2 -7070.527} C_VEL
LIN {X 0,Y 482.777,Z 389.418,A -85,B 0,C 180,E1 -7070.854,E2 -7070.854} C_VEL
LIN {X 0,Y 482.545,Z 398.646,A -85,B 0,C 180,E1 -7071.323,E2 -7071.323} C_VEL
LIN {X 0,Y 482.271,Z 408.481,A -85,B 0,C 180,E1 -7071.973,E2 -7071.973} C_VEL
LIN {X 0,Y 481.918,Z 417.613,A -85,B 0,C 180,E1 -7072.757,E2 -7072.757} C_VEL
LIN {X 0,Y 481.658,Z 425.154,A -85,B 0,C 180,E1 -7073.57,E2 -7073.57} C_VEL
LIN {X 0,Y 481.597,Z 427.528,A -85,B 0,C 180,E1 -7073.864,E2 -7073.864} C_VEL
LIN {X 0,Y 480.842,Z 431.533,A -85,B 0,C 180,E1 -7074.377,E2 -7074.377} C_VEL
LIN {X 0,Y 477.775,Z 437.525,A -85,B 0,C 180,E1 -7075.252,E2 -7075.252} C_VEL
LIN {X 0,Y 474.699,Z 442.638,A -85,B 0,C 180,E1 -7076.209,E2 -7076.209} C_VEL
LIN {X 0,Y 473.939,Z 445.242,A -85,B 0,C 180,E1 -7076.845,E2 -7076.845} C_VEL
LIN {X 0,Y 473.909,Z 448.407,A -85,B 0,C 180,E1 -7077.734,E2 -7077.734} C_VEL
LIN {X 0,Y 473.814,Z 451.116,A -85,B 0,C 180,E1 -7078.726,E2 -7078.726} C_VEL
LIN {X 0,Y 473.727,Z 453.042,A -85,B 0,C 180,E1 -7079.709,E2 -7079.709} C_VEL
LIN {X 0,Y 473.621,Z 454.617,A -85,B 0,C 180,E1 -7081.104,E2 -7081.104} C_VEL
LIN {X 0,Y 473.589,Z 454.748,A -85,B 0,C 180,E1 -7082.612,E2 -7082.612} C_VEL
LIN {X 0,Y 473.618,Z 454.059,A -85,B 0,C 180,E1 -7083.567,E2 -7083.567} C_VEL
LIN {X 0,Y 473.706,Z 452.164,A -85,B 0,C 180,E1 -7084.825,E2 -7084.825} C_VEL
LIN {X 0,Y 473.84,Z 449.542,A -85,B 0,C 180,E1 -7085.929,E2 -7085.929} C_VEL
LIN {X 0,Y 473.928,Z 446.633,A -85,B 0,C 180,E1 -7086.841,E2 -7086.841} C_VEL
LIN {X 0,Y 474.027,Z 442.845,A -85,B 0,C 180,E1 -7087.787,E2 -7087.787} C_VEL
LIN {X 0,Y 474.169,Z 438.475,A -85,B 0,C 180,E1 -7088.675,E2 -7088.675} C_VEL
LIN {X 0,Y 474.384,Z 432.759,A -85,B 0,C 180,E1 -7089.626,E2 -7089.626} C_VEL
LIN {X 0,Y 474.61,Z 426.052,A -85,B 0,C 180,E1 -7090.539,E2 -7090.539} C_VEL
LIN {X 0,Y 474.896,Z 418.317,A -85,B 0,C 180,E1 -7091.398,E2 -7091.398} C_VEL
LIN {X 0,Y 475.24,Z 408.789,A -85,B 0,C 180,E1 -7092.242,E2 -7092.242} C_VEL
LIN {X 0,Y 475.561,Z 398.67,A -85,B 0,C 180,E1 -7092.92,E2 -7092.92} C_VEL
LIN {X 0,Y 475.776,Z 389.995,A -85,B 0,C 180,E1 -7093.37,E2 -7093.37} C_VEL
LIN {X 0,Y 475.923,Z 380.59,A -85,B 0,C 180,E1 -7093.734,E2 -7093.734} C_VEL
LIN {X 0,Y 476.104,Z 371.982,A -85,B 0,C 180,E1 -7093.96,E2 -7093.96} C_VEL
LIN {X 0,Y 476.433,Z 307.732,A -85,B 0,C 180,E1 -7094.958,E2 -7094.958} C_VEL
LIN {X 0,Y 474.563,Z 296.132,A -85,B 0,C 180,E1 -7095.199,E2 -7095.199} C_VEL
LIN {X 0,Y 474.894,Z 282.325,A -85,B 0,C 180,E1 -7098.476,E2 -7098.476} C_VEL
LIN {X 0,Y 474.991,Z 273.354,A -85,B 0,C 180,E1 -7100.633,E2 -7100.633} C_VEL
LIN {X 0,Y 474.79,Z 271.159,A -85,B 0,C 180,E1 -7101.22,E2 -7101.22} C_VEL
LIN {X 0,Y 474.772,Z 271.158,A -85,B 0,C 180,E1 -7104.053,E2 -7104.053} C_VEL
LIN {X 0,Y 474.895,Z 271.141,A -85,B 0,C 180,E1 -7107.455,E2 -7107.455} C_VEL
LIN {X 0,Y 474.914,Z 271.143,A -85,B 0,C 180,E1 -7110,E2 -7110} C_VEL
LIN {X 0,Y 474.896,Z 271.139,A -85,B 0,C 180,E1 -7112.545,E2 -7112.545} C_VEL
LIN {X 0,Y 474.76,Z 271.16,A -85,B 0,C 180,E1 -7115.948,E2 -7115.948} C_VEL
LIN {X 0,Y 474.728,Z 271.162,A -85,B 0,C 180,E1 -7118.513,E2 -7118.513} C_VEL
LIN {X 0,Y 474.706,Z 271.164,A -85,B 0,C 180,E1 -7121.962,E2 -7121.962} C_VEL
LIN {X 0,Y 474.701,Z 271.161,A -85,B 0,C 180,E1 -7125.455,E2 -7125.455} C_VEL
LIN {X 0,Y 474.663,Z 271.169,A -85,B 0,C 180,E1 -7129.01,E2 -7129.01} C_VEL
LIN {X 0,Y 474.588,Z 271.175,A -85,B 0,C 180,E1 -7131.728,E2 -7131.728} C_VEL
LIN {X 0,Y 474.654,Z 271.172,A -85,B 0,C 180,E1 -7134.492,E2 -7134.492} C_VEL
LIN {X 0,Y 474.68,Z 271.167,A -85,B 0,C 180,E1 -7137.334,E2 -7137.334} C_VEL
LIN {X 0,Y 474.603,Z 271.174,A -85,B 0,C 180,E1 -7140.229,E2 -7140.229} C_VEL
LIN {X 0,Y 474.621,Z 271.178,A -85,B 0,C 180,E1 -7143.221,E2 -7143.221} C_VEL
LIN {X 0,Y 474.584,Z 271.176,A -85,B 0,C 180,E1 -7146.323,E2 -7146.323} C_VEL
LIN {X 0,Y 474.622,Z 271.175,A -85,B 0,C 180,E1 -7149.647,E2 -7149.647} C_VEL
LIN {X 0,Y 474.609,Z 271.175,A -85,B 0,C 180,E1 -7152.933,E2 -7152.933} C_VEL
LIN {X 0,Y 474.612,Z 271.176,A -85,B 0,C 180,E1 -7155.895,E2 -7155.895} C_VEL
LIN {X 0,Y 474.639,Z 271.17,A -85,B 0,C 180,E1 -7159.037,E2 -7159.037} C_VEL
LIN {X 0,Y 474.609,Z 271.181,A -85,B 0,C 180,E1 -7161.702,E2 -7161.702} C_VEL
LIN {X 0,Y 474.621,Z 271.171,A -85,B 0,C 180,E1 -7164.725,E2 -7164.725} C_VEL
LIN {X 0,Y 474.627,Z 271.177,A -85,B 0,C 180,E1 -7167.787,E2 -7167.787} C_VEL
LIN {X 0,Y 474.622,Z 271.171,A -85,B 0,C 180,E1 -7170.882,E2 -7170.882} C_VEL
LIN {X 0,Y 474.656,Z 271.169,A -85,B 0,C 180,E1 -7173.628,E2 -7173.628} C_VEL
LIN {X 0,Y 474.625,Z 271.174,A -85,B 0,C 180,E1 -7176.641,E2 -7176.641} C_VEL
LIN {X 0,Y 474.643,Z 271.173,A -85,B 0,C 180,E1 -7180.089,E2 -7180.089} C_VEL
LIN {X 0,Y 474.638,Z 271.174,A -85,B 0,C 180,E1 -7182.774,E2 -7182.774} C_VEL
LIN {X 0,Y 474.635,Z 271.169,A -85,B 0,C 180,E1 -7185.42,E2 -7185.42} C_VEL
LIN {X 0,Y 474.691,Z 271.163,A -85,B 0,C 180,E1 -7188.037,E2 -7188.037} C_VEL
LIN {X 0,Y 474.715,Z 271.16,A -85,B 0,C 180,E1 -7191.486,E2 -7191.486} C_VEL
LIN {X 0,Y 474.757,Z 271.154,A -85,B 0,C 180,E1 -7194.052,E2 -7194.052} C_VEL
LIN {X 0,Y 474.88,Z 271.142,A -85,B 0,C 180,E1 -7197.455,E2 -7197.455} C_VEL
LIN {X 0,Y 474.864,Z 271.146,A -85,B 0,C 180,E1 -7200.848,E2 -7200.848} C_VEL
LIN {X 0,Y 474.88,Z 271.14,A -85,B 0,C 180,E1 -7202.545,E2 -7202.545} C_VEL
LIN {X 0,Y 474.761,Z 271.155,A -85,B 0,C 180,E1 -7205.948,E2 -7205.948} C_VEL
LIN {X 0,Y 474.715,Z 271.159,A -85,B 0,C 180,E1 -7208.514,E2 -7208.514} C_VEL
LIN {X 0,Y 474.727,Z 271.161,A -85,B 0,C 180,E1 -7211.962,E2 -7211.962} C_VEL
LIN {X 0,Y 474.668,Z 271.173,A -85,B 0,C 180,E1 -7215.768,E2 -7215.768} C_VEL
LIN {X 0,Y 474.652,Z 271.168,A -85,B 0,C 180,E1 -7219.011,E2 -7219.011} C_VEL
LIN {X 0,Y 474.577,Z 271.184,A -85,B 0,C 180,E1 -7221.729,E2 -7221.729} C_VEL
LIN {X 0,Y 474.647,Z 271.17,A -85,B 0,C 180,E1 -7224.493,E2 -7224.493} C_VEL
LIN {X 0,Y 474.669,Z 271.166,A -85,B 0,C 180,E1 -7227.335,E2 -7227.335} C_VEL
LIN {X 0,Y 474.593,Z 271.176,A -85,B 0,C 180,E1 -7230.811,E2 -7230.811} C_VEL
LIN {X 0,Y 474.628,Z 271.174,A -85,B 0,C 180,E1 -7233.985,E2 -7233.985} C_VEL
LIN {X 0,Y 474.564,Z 271.181,A -85,B 0,C 180,E1 -7236.9,E2 -7236.9} C_VEL
LIN {X 0,Y 474.608,Z 271.173,A -85,B 0,C 180,E1 -7239.647,E2 -7239.647} C_VEL
LIN {X 0,Y 474.606,Z 271.177,A -85,B 0,C 180,E1 -7242.935,E2 -7242.935} C_VEL
LIN {X 0,Y 474.596,Z 271.174,A -85,B 0,C 180,E1 -7245.895,E2 -7245.895} C_VEL
LIN {X 0,Y 474.614,Z 271.178,A -85,B 0,C 180,E1 -7249.043,E2 -7249.043} C_VEL
LIN {X 0,Y 474.603,Z 271.174,A -85,B 0,C 180,E1 -7251.705,E2 -7251.705} C_VEL
LIN {X 0,Y 474.617,Z 271.176,A -85,B 0,C 180,E1 -7254.726,E2 -7254.726} C_VEL
LIN {X 0,Y 474.63,Z 271.171,A -85,B 0,C 180,E1 -7257.788,E2 -7257.788} C_VEL
LIN {X 0,Y 474.602,Z 271.177,A -85,B 0,C 180,E1 -7260.889,E2 -7260.889} C_VEL
LIN {X 0,Y 474.59,Z 271.182,A -85,B 0,C 180,E1 -7263.625,E2 -7263.625} C_VEL
LIN {X 0,Y 474.67,Z 271.314,A -85,B 0,C 180,E1 -7266.632,E2 -7266.632} C_VEL
LIN {X 0,Y 475.867,Z 279.145,A -85,B 0,C 180,E1 -7268.333,E2 -7268.333} C_VEL
LIN {X 0,Y 475.277,Z 294.621,A -85,B 0,C 180,E1 -7271.517,E2 -7271.517} C_VEL
LIN {X 0,Y 474.79,Z 309.558,A -85,B 0,C 180,E1 -7274.548,E2 -7274.548} C_VEL
LIN {X 0,Y 474.476,Z 320.931,A -85,B 0,C 180,E1 -7276.833,E2 -7276.833} C_VEL
LIN {X 0,Y 476.408,Z 336.656,A -85,B 0,C 180,E1 -7277.132,E2 -7277.132} C_VEL
LIN {X 0,Y 476.058,Z 397.378,A -85,B 0,C 180,E1 -7278.072,E2 -7278.072} C_VEL
LIN {X 0,Y 475.808,Z 406.538,A -85,B 0,C 180,E1 -7278.309,E2 -7278.309} C_VEL
LIN {X 0,Y 475.613,Z 415.576,A -85,B 0,C 180,E1 -7278.655,E2 -7278.655} C_VEL
LIN {X 0,Y 475.325,Z 424.868,A -85,B 0,C 180,E1 -7279.134,E2 -7279.134} C_VEL
LIN {X 0,Y 475.085,Z 434.43,A -85,B 0,C 180,E1 -7279.775,E2 -7279.775} C_VEL
LIN {X 0,Y 474.725,Z 444.183,A -85,B 0,C 180,E1 -7280.628,E2 -7280.628} C_VEL
LIN {X 0,Y 474.411,Z 451.926,A -85,B 0,C 180,E1 -7281.481,E2 -7281.481} C_VEL
LIN {X 0,Y 474.191,Z 458.302,A -85,B 0,C 180,E1 -7282.335,E2 -7282.335} C_VEL
LIN {X 0,Y 474.072,Z 463.602,A -85,B 0,C 180,E1 -7283.189,E2 -7283.189} C_VEL
LIN {X 0,Y 473.961,Z 468.02,A -85,B 0,C 180,E1 -7284.042,E2 -7284.042} C_VEL
LIN {X 0,Y 473.793,Z 473.221,A -85,B 0,C 180,E1 -7285.321,E2 -7285.321} C_VEL
LIN {X 0,Y 473.816,Z 475.886,A -85,B 0,C 180,E1 -7286.173,E2 -7286.173} C_VEL
LIN {X 0,Y 473.745,Z 478.803,A -85,B 0,C 180,E1 -7287.449,E2 -7287.449} C_VEL
LIN {X 0,Y 473.696,Z 480.063,A -85,B 0,C 180,E1 -7288.3,E2 -7288.3} C_VEL
LIN {X 0,Y 473.686,Z 480.847,A -85,B 0,C 180,E1 -7289.15,E2 -7289.15} C_VEL
LIN {X 0,Y 473.668,Z 481.141,A -85,B 0,C 180,E1 -7290,E2 -7290} C_VEL
LIN {X 0,Y 473.685,Z 480.842,A -85,B 0,C 180,E1 -7290.85,E2 -7290.85} C_VEL
LIN {X 0,Y 473.696,Z 480.056,A -85,B 0,C 180,E1 -7291.7,E2 -7291.7} C_VEL
LIN {X 0,Y 473.745,Z 478.795,A -85,B 0,C 180,E1 -7292.551,E2 -7292.551} C_VEL
LIN {X 0,Y 473.816,Z 475.873,A -85,B 0,C 180,E1 -7293.827,E2 -7293.827} C_VEL
LIN {X 0,Y 473.793,Z 473.209,A -85,B 0,C 180,E1 -7294.679,E2 -7294.679} C_VEL
LIN {X 0,Y 473.947,Z 468.001,A -85,B 0,C 180,E1 -7295.958,E2 -7295.958} C_VEL
LIN {X 0,Y 474.122,Z 461.137,A -85,B 0,C 180,E1 -7297.238,E2 -7297.238} C_VEL
LIN {X 0,Y 474.34,Z 453.636,A -85,B 0,C 180,E1 -7298.306,E2 -7298.306} C_VEL
